			3:
				IF	(* Zylinder ist ausgefahren *)
					(e_sensor1_ausgefahren AND NOT e_sensor1_eingefahren AND NOT e_sensor_mittegefahren) OR
					(* Zylinder steht in Mittelstellung *)
					(e_sensor_mittegefahren AND NOT e_sensor1_eingefahren AND NOT e_sensor1_ausgefahren)
					THEN
						fb_state_entry.i16_next_step := AUSGEFAHREN;
				ELSE
					IF i16_betriebsart <> HAND AND st_config.b_aktiv THEN
						(* Zeitüberwachung *)
						IF fb_ton_uz_fahren.Q AND (NOT b_nockengesteuert OR b_no_gesteuert_im_norm_betrieb) THEN
							st_sm.b_zeit_ausfahren1 := TRUE;
							fb_state_entry.i16_next_step := ZYL_FEHLER;
						(* Winkelüberwachung *)
						ELSIF uw_nocken_zylinder_ausfahren AND b_nockengesteuert AND NOT b_no_gesteuert_im_norm_betrieb AND NOT b_zustand_uw_nocken_ausfahren THEN
							st_sm.b_winkel_ausfahren1 := TRUE;
							fb_state_entry.i16_next_step := ZYL_FEHLER;
						END_IF
					END_IF
				END_IF
				IF i16_betriebsart <> HAND AND st_config.b_aktiv THEN
					(* Überwachung auf Sensorfehler *)
					IF e_sensor1_ausgefahren  AND e_sensor1_eingefahren  AND st_config.b_sensor1_aktiv THEN
						fb_ton_uz_sensor1.IN := TRUE;
						IF fb_ton_uz_sensor1.Q THEN
							st_sm.b_sensor1 := TRUE;
							fb_state_entry.i16_next_step := ZYL_FEHLER;
						END_IF
					ELSE
						fb_ton_uz_sensor1.IN := FALSE;
					END_IF
				END_IF

			4:
				IF e_sensor1_ausgefahren AND e_sensor2_ausgefahren AND NOT e_sensor1_eingefahren AND NOT e_sensor2_eingefahren	THEN
					fb_state_entry.i16_next_step := AUSGEFAHREN;
				ELSE
					IF i16_betriebsart <> HAND AND st_config.b_aktiv THEN
						IF NOT e_sensor1_ausgefahren OR NOT e_sensor2_ausgefahren THEN
							(* Zeitüberwachung *)
							IF fb_ton_uz_fahren.Q AND (NOT b_nockengesteuert OR b_no_gesteuert_im_norm_betrieb) THEN
								IF NOT e_sensor1_ausgefahren THEN
									st_sm.b_zeit_ausfahren1 := TRUE;
								END_IF
								IF NOT e_sensor2_ausgefahren THEN
									st_sm.b_zeit_ausfahren2 := TRUE;
								END_IF
								fb_state_entry.i16_next_step := ZYL_FEHLER;
							(* Winkelüberwachung *)
							ELSIF uw_nocken_zylinder_ausfahren AND b_nockengesteuert AND NOT b_no_gesteuert_im_norm_betrieb AND NOT b_zustand_uw_nocken_ausfahren THEN
								IF NOT e_sensor1_ausgefahren THEN
									st_sm.b_winkel_ausfahren1 := TRUE;
								END_IF
								IF NOT e_sensor2_ausgefahren THEN
									st_sm.b_winkel_ausfahren2 := TRUE;
								END_IF
								fb_state_entry.i16_next_step := ZYL_FEHLER;
							END_IF
						END_IF
					END_IF
				END_IF

				IF i16_betriebsart <> HAND AND st_config.b_aktiv THEN
					(* Überwachung auf Sensorfehler *)
					IF e_sensor1_ausgefahren  AND e_sensor1_eingefahren  AND st_config.b_sensor1_aktiv THEN
						fb_ton_uz_sensor1.IN := TRUE;
						IF fb_ton_uz_sensor1.Q THEN
							st_sm.b_sensor1 := TRUE;
							fb_state_entry.i16_next_step := ZYL_FEHLER;
						END_IF
					ELSE
						fb_ton_uz_sensor1.IN := FALSE;
					END_IF
					IF e_sensor2_ausgefahren  AND e_sensor2_eingefahren  AND st_config.b_sensor2_aktiv THEN
						fb_ton_uz_sensor2.IN := TRUE;
						IF fb_ton_uz_sensor2.Q THEN
							st_sm.b_sensor2 := TRUE;
							fb_state_entry.i16_next_step := ZYL_FEHLER;
						END_IF
					ELSE
						fb_ton_uz_sensor2.IN := FALSE;
					END_IF
				END_IF

			6:
				IF 	e_sensor1_ausgefahren AND
					e_sensor2_ausgefahren AND
					e_sensor3_ausgefahren AND
					NOT e_sensor1_eingefahren AND
					NOT e_sensor2_eingefahren AND
					NOT e_sensor3_eingefahren
					THEN
						fb_state_entry.i16_next_step := AUSGEFAHREN;
				ELSE
					IF i16_betriebsart <> HAND AND st_config.b_aktiv THEN
						IF NOT e_sensor1_ausgefahren OR NOT e_sensor2_ausgefahren OR NOT e_sensor3_ausgefahren THEN
							(* Zeitüberwachung *)
							IF fb_ton_uz_fahren.Q AND (NOT b_nockengesteuert OR b_no_gesteuert_im_norm_betrieb) THEN
								IF NOT e_sensor1_ausgefahren THEN
									st_sm.b_zeit_ausfahren1 := TRUE;
								END_IF
								IF NOT e_sensor2_ausgefahren THEN
									st_sm.b_zeit_ausfahren2 := TRUE;
								END_IF
								IF NOT e_sensor3_ausgefahren THEN
									st_sm.b_zeit_ausfahren3 := TRUE;
								END_IF
								fb_state_entry.i16_next_step := ZYL_FEHLER;
							(* Winkelüberwachung *)
							ELSIF uw_nocken_zylinder_ausfahren AND b_nockengesteuert AND NOT b_no_gesteuert_im_norm_betrieb AND NOT b_zustand_uw_nocken_ausfahren THEN
								IF NOT e_sensor1_ausgefahren THEN
									st_sm.b_winkel_ausfahren1 := TRUE;
								END_IF
								IF NOT e_sensor2_ausgefahren THEN
									st_sm.b_winkel_ausfahren2 := TRUE;
								END_IF
								IF NOT e_sensor3_ausgefahren THEN
									st_sm.b_winkel_ausfahren3 := TRUE;
								END_IF
								fb_state_entry.i16_next_step := ZYL_FEHLER;
							END_IF
						END_IF
					END_IF
				END_IF

				IF i16_betriebsart <> HAND AND st_config.b_aktiv THEN
					(* Überwachung auf Sensorfehler *)
					IF e_sensor1_ausgefahren  AND e_sensor1_eingefahren  AND st_config.b_sensor1_aktiv THEN
						fb_ton_uz_sensor1.IN := TRUE;
						IF fb_ton_uz_sensor1.Q THEN
							st_sm.b_sensor1 := TRUE;
							fb_state_entry.i16_next_step := ZYL_FEHLER;
						END_IF
					ELSE
						fb_ton_uz_sensor1.IN := FALSE;
					END_IF
					IF e_sensor2_ausgefahren  AND e_sensor2_eingefahren  AND st_config.b_sensor2_aktiv THEN
						fb_ton_uz_sensor2.IN := TRUE;
						IF fb_ton_uz_sensor2.Q THEN
							st_sm.b_sensor2 := TRUE;
							fb_state_entry.i16_next_step := ZYL_FEHLER;
						END_IF
					ELSE
						fb_ton_uz_sensor2.IN := FALSE;
					END_IF
					IF e_sensor3_ausgefahren  AND e_sensor3_eingefahren  AND st_config.b_sensor3_aktiv THEN
						fb_ton_uz_sensor3.IN := TRUE;
						IF fb_ton_uz_sensor3.Q THEN
							st_sm.b_sensor3 := TRUE;
							fb_state_entry.i16_next_step := ZYL_FEHLER;
						END_IF
					ELSE
						fb_ton_uz_sensor3.IN := FALSE;
					END_IF
				END_IF
		END_CASE

(*=======================================================*)
	AUSGEFAHREN:
		IF fb_state_entry.E THEN
			st_ctrl_out.b_gestoppt := FALSE;
			st_ctrl_out.b_eingefahren := FALSE;
			st_ctrl_out.b_ohne_luft := FALSE;
			fb_ton_einausfahren.IN := FALSE;
			fb_ton_uz_fahren.IN := FALSE;
			fb_ton_uz_sensor1.IN := FALSE;
			fb_ton_uz_sensor2.IN := FALSE;
			fb_ton_uz_sensor3.IN := FALSE;
			st_tzk.fb_ton_tzk.IN := FALSE;
			a_ventil_ausfahren := TRUE;
			b_zustand_uw_nocken_ausfahren := FALSE;
			IF NOT b_mit_tzk THEN
				st_ctrl_out.b_ausgefahren := TRUE;
			END_IF
		END_IF

		IF st_ctrl_in.b_ausfahren THEN	(* Messagewiederholung wenn der Zylinder sich schon im gewünschten Zustand befindet*)
			st_ctrl_out.b_ausgefahren := TRUE;
		END_IF

		(*-----------------------Weiterschaltbedingungen----------------------------*)
		CASE i16_betriebsart OF
		KEINE:
			;
		AUTO, TIPPEN, DUMMY, PSEUDO:
			IF	(st_ctrl_in.b_einfahren AND
				NOT bw_nocken_zylinder_einfahren AND
				NOT b_ibn_zylinder_einfahren AND
				NOT b_direkttaste_einfahren AND
				NOT e_taste_einfahren) OR
				(NOT st_ctrl_in.b_einfahren AND
				bw_nocken_zylinder_einfahren AND
				NOT b_ibn_zylinder_einfahren AND
				NOT b_direkttaste_einfahren AND
				NOT e_taste_einfahren) OR
				(NOT st_ctrl_in.b_einfahren AND
				NOT bw_nocken_zylinder_einfahren AND
				b_ibn_zylinder_einfahren AND
				NOT b_direkttaste_einfahren AND
				NOT e_taste_einfahren)
				THEN
					IF i16_anzahl_sensoren >= 1AND b_sensor_eingefahren_vorhanden AND b_mit_tzk THEN
						st_tzk.t_einfahrzeit_kompensiert := (st_tzk.t_einfahrzeit * st_config.i16_tzk_faktor_einfahren) / 100;
					END_IF
					fb_state_entry.i16_next_step := BEWEGUNG_EINFAHREN;

			ELSIF	st_ctrl_in.b_luftlos AND
					NOT bw_nocken_zylinder_einfahren AND
					NOT b_ibn_zylinder_einfahren AND
					NOT b_direkttaste_einfahren AND
					NOT e_taste_einfahren AND
					NOT bw_nocken_zylinder_ausfahren AND
					NOT b_ibn_zylinder_ausfahren AND
					NOT b_direkttaste_ausfahren AND
					NOT e_taste_ausfahren
					THEN
						fb_state_entry.i16_next_step := LUFTLOS;
			END_IF
		HAND:
			IF	(st_visu.i16_nr_zyl_im_handbetrieb = st_config.i16_identnummer AND (st_visu.b_taste_einfahren OR e_taste_einfahren)) OR
				(bw_nocken_zylinder_einfahren AND b_nockengesteuert AND b_masterachse_hand_dialog_aktiv)
				THEN
					IF i16_anzahl_sensoren >= 1AND b_sensor_eingefahren_vorhanden AND b_mit_tzk THEN
						st_tzk.t_einfahrzeit_kompensiert := (st_tzk.t_einfahrzeit * st_config.i16_tzk_faktor_einfahren) / 100;
					END_IF
					fb_state_entry.i16_next_step := BEWEGUNG_EINFAHREN;
			END_IF
		END_CASE

		(* Überwachung auf Endlagenfehler *)
		IF i16_betriebsart <> HAND AND st_config.b_aktiv THEN
			CASE i16_anzahl_sensoren OF
				1,2,3:	(* Alle Zylinder mit mindestens einem Sensor für EINGEFAHREN *)
					IF b_sensor_ausgefahren_vorhanden AND st_config.b_endlage1_aktiv AND NOT e_sensor1_ausgefahren THEN
						fb_ton_uz_endlage1.IN := TRUE;
						IF fb_ton_uz_endlage1.Q THEN
							st_sm.b_endlage1 := TRUE;
							fb_state_entry.i16_next_step := ZYL_FEHLER;
						END_IF
					ELSE
						fb_ton_uz_endlage1.IN := FALSE;
					END_IF

				4:	(* Alle Zylinder mit 2 Sensoren für EINGEFAHREN *)
					IF b_sensor_ausgefahren_vorhanden AND st_config.b_endlage1_aktiv AND NOT e_sensor1_ausgefahren THEN
						fb_ton_uz_endlage1.IN := TRUE;
						IF fb_ton_uz_endlage1.Q THEN
							st_sm.b_endlage1 := TRUE;
							fb_state_entry.i16_next_step := ZYL_FEHLER;
						END_IF
					ELSE
						fb_ton_uz_endlage1.IN := FALSE;
					END_IF
					IF b_sensor_ausgefahren_vorhanden AND st_config.b_endlage2_aktiv AND NOT e_sensor2_ausgefahren THEN
						fb_ton_uz_endlage2.IN := TRUE;
						IF fb_ton_uz_endlage2.Q THEN
							st_sm.b_endlage2 := TRUE;
							fb_state_entry.i16_next_step := ZYL_FEHLER;
						END_IF
					ELSE
						fb_ton_uz_endlage2.IN := FALSE;
					END_IF

				6:	(* Alle Zylinder mit 3 Sensoren für EINGEFAHREN *)
					IF b_sensor_ausgefahren_vorhanden AND st_config.b_endlage1_aktiv AND NOT e_sensor1_ausgefahren THEN
						fb_ton_uz_endlage1.IN := TRUE;
						IF fb_ton_uz_endlage1.Q THEN
							st_sm.b_endlage1 := TRUE;
							fb_state_entry.i16_next_step := ZYL_FEHLER;
						END_IF
					ELSE
						fb_ton_uz_endlage1.IN := FALSE;
					END_IF
					IF b_sensor_ausgefahren_vorhanden AND st_config.b_endlage2_aktiv AND NOT e_sensor2_ausgefahren THEN
						fb_ton_uz_endlage2.IN := TRUE;
						IF fb_ton_uz_endlage2.Q THEN
							st_sm.b_endlage2 := TRUE;
							fb_state_entry.i16_next_step := ZYL_FEHLER;
						END_IF
					ELSE
						fb_ton_uz_endlage2.IN := FALSE;
					END_IF
					IF b_sensor_ausgefahren_vorhanden AND st_config.b_endlage3_aktiv AND NOT e_sensor3_ausgefahren THEN
						fb_ton_uz_endlage3.IN := TRUE;
						IF fb_ton_uz_endlage3.Q THEN
							st_sm.b_endlage3 := TRUE;
							fb_state_entry.i16_next_step := ZYL_FEHLER;
						END_IF
					ELSE
						fb_ton_uz_endlage3.IN := FALSE;
					END_IF
			END_CASE
		END_IF

(*=======================================================*)
	BEWEGUNG_EINFAHREN:
		IF fb_state_entry.E THEN
			st_ctrl_out.b_gestoppt := FALSE;
			st_ctrl_out.b_eingefahren := FALSE;
			st_ctrl_out.b_ausgefahren := FALSE;
			st_ctrl_out.b_ohne_luft := FALSE;
			st_ctrl_out.b_fehler := FALSE;
			a_ventil_ausfahren := FALSE;
			a_ventil_einfahren := TRUE;
			fb_ton_uz_fahren.IN := TRUE;
			fb_ton_einausfahren.IN := TRUE;
			fb_ton_uz_endlage1.IN := FALSE;
			fb_ton_uz_endlage2.IN := FALSE;
			fb_ton_uz_endlage3.IN := FALSE;
			st_sm.b_zeit_ausfahren1:= FALSE;
			st_sm.b_zeit_einfahren1:= FALSE;
			st_sm.b_endlage1	:= FALSE;
			st_sm.b_sensor1:= FALSE;
			st_sm.b_zeit_ausfahren2 := FALSE;
			st_sm.b_zeit_einfahren2 := FALSE;
			st_sm.b_endlage2	:= FALSE;
			st_sm.b_sensor2 := FALSE;
			st_sm.b_zeit_ausfahren3 := FALSE;
			st_sm.b_zeit_einfahren3 := FALSE;
			st_sm.b_endlage3	:= FALSE;
			st_sm.b_sensor3 := FALSE;
			st_sm.b_winkel_ausfahren1:= FALSE;
			st_sm.b_winkel_einfahren1:= FALSE;
			st_sm.b_winkel_ausfahren2 := FALSE;
			st_sm.b_winkel_einfahren2 := FALSE;
			st_sm.b_winkel_ausfahren3 := FALSE;
			st_sm.b_winkel_einfahren3 := FALSE;
			st_sm.b_zyltyp_nicht_definiert := FALSE;
			st_sm.b_reserve1:= FALSE;
			(* Verhindere die sofortige Fehlerauslösung, wenn Überwachungsnocken bei Stateentry schon vorhanden ist *)
			IF uw_nocken_zylinder_einfahren THEN
				b_zustand_uw_nocken_einfahren := TRUE;
			END_IF
		END_IF

		(* Fehlermeldung für nockengesteuerte Zylinder wieder freischalten *)
		IF fb_ton_uz_fahren.Q THEN
			b_zustand_uw_nocken_einfahren := FALSE;
		END_IF

		CASE i16_betriebsart OF
		KEINE:
			;
		AUTO, TIPPEN, DUMMY, PSEUDO:
			IF 	(st_ctrl_in.b_ausfahren AND
				NOT bw_nocken_zylinder_ausfahren AND
				NOT b_ibn_zylinder_ausfahren AND
				NOT b_direkttaste_ausfahren AND
				NOT e_taste_ausfahren) OR
				(NOT st_ctrl_in.b_ausfahren AND
				bw_nocken_zylinder_ausfahren AND
				NOT b_ibn_zylinder_ausfahren AND
				NOT b_direkttaste_ausfahren AND
				NOT e_taste_ausfahren) OR
				(NOT st_ctrl_in.b_ausfahren AND
				NOT bw_nocken_zylinder_ausfahren AND
				b_ibn_zylinder_ausfahren AND
				NOT b_direkttaste_ausfahren AND
				NOT e_taste_ausfahren)
				THEN
					IF i16_anzahl_sensoren >= 1AND b_sensor_ausgefahren_vorhanden AND b_mit_tzk THEN
						st_tzk.t_ausfahrzeit_kompensiert := (st_tzk.t_ausfahrzeit * st_config.i16_tzk_faktor_ausfahren) / 100;
					END_IF
					fb_state_entry.i16_next_step := BEWEGUNG_AUSFAHREN;
			END_IF
		HAND:
			IF	(st_visu.i16_nr_zyl_im_handbetrieb = st_config.i16_identnummer AND (st_visu.b_taste_ausfahren OR e_taste_ausfahren)) OR
				(bw_nocken_zylinder_ausfahren AND b_nockengesteuert AND b_masterachse_hand_dialog_aktiv)
				THEN
					IF i16_anzahl_sensoren >= 1AND b_sensor_ausgefahren_vorhanden AND b_mit_tzk THEN
						st_tzk.t_ausfahrzeit_kompensiert := (st_tzk.t_ausfahrzeit * st_config.i16_tzk_faktor_ausfahren) / 100;
					END_IF
					fb_state_entry.i16_next_step := BEWEGUNG_AUSFAHREN;
			END_IF
		END_CASE

		(* Totzeitkompensation mit Plausibilitätscheck der ermittelten Kompensationszeit *)
		IF 	i16_anzahl_sensoren >= 1AND
			b_sensor_eingefahren_vorhanden AND
			b_mit_tzk AND
			st_tzk.t_einfahrzeit_kompensiert < st_tzk.t_einfahrzeit
			THEN
				st_tzk.fb_ton_tzk.PT := st_tzk.t_einfahrzeit_kompensiert ;
				st_tzk.fb_ton_tzk.IN := TRUE;
				(* Totzeit ist abgelaufen -> vorzeitig "eingefahren" melden*)
				IF st_tzk.fb_ton_tzk.Q THEN
					st_tzk.fb_ton_tzk.IN := FALSE;
					st_ctrl_out.b_eingefahren := TRUE;
				END_IF
		END_IF

		(*-----------------------Weiterschaltbedingungen----------------------------*)
		(* Bedingungen für Zylinder ist eingefahren und Fehlervorkommen*)
		(* Die Sensorkonfiguration "vorhanden" ist nur für die Fälle 1, 2 von Bedeutung wegen Sonderzylinder *)
		CASE i16_anzahl_sensoren OF
			0:
				IF fb_ton_einausfahren.Q THEN
					fb_state_entry.i16_next_step := EINGEFAHREN;
				END_IF

			1:
				IF b_sensor_eingefahren_vorhanden THEN
					IF e_sensor1_eingefahren THEN
						fb_state_entry.i16_next_step := EINGEFAHREN;
					ELSE
						IF i16_betriebsart <> HAND AND st_config.b_aktiv THEN
							(* Zeitüberwachung *)
							IF fb_ton_uz_fahren.Q AND (NOT b_nockengesteuert OR b_no_gesteuert_im_norm_betrieb)THEN
								st_sm.b_zeit_einfahren1 := TRUE;
								fb_state_entry.i16_next_step := ZYL_FEHLER;
							(* Winkelüberwachung *)
							ELSIF uw_nocken_zylinder_einfahren AND b_nockengesteuert AND NOT b_no_gesteuert_im_norm_betrieb AND NOT b_zustand_uw_nocken_einfahren THEN
								st_sm.b_winkel_einfahren1 := TRUE;
								fb_state_entry.i16_next_step := ZYL_FEHLER;
							END_IF
						END_IF
					END_IF
				ELSIF b_sensor_ausgefahren_vorhanden THEN
					IF  NOT e_sensor1_ausgefahren THEN
						fb_state_entry.i16_next_step := EINGEFAHREN;
					ELSE
						IF i16_betriebsart <> HAND AND st_config.b_aktiv THEN
							(* Zeitüberwachung *)
							IF fb_ton_uz_fahren.Q AND (NOT b_nockengesteuert OR b_no_gesteuert_im_norm_betrieb)THEN
								st_sm.b_zeit_einfahren1 := TRUE;
								fb_state_entry.i16_next_step := ZYL_FEHLER;
							(* Winkelüberwachung *)
							ELSIF uw_nocken_zylinder_einfahren AND b_nockengesteuert AND NOT b_no_gesteuert_im_norm_betrieb AND NOT b_zustand_uw_nocken_einfahren THEN
								st_sm.b_winkel_einfahren1 := TRUE;
								fb_state_entry.i16_next_step := ZYL_FEHLER;
							END_IF
						END_IF
					END_IF
				END_IF

			2:
				IF b_sensor_eingefahren_vorhanden AND b_sensor_ausgefahren_vorhanden THEN
					IF e_sensor1_eingefahren AND NOT e_sensor1_ausgefahren THEN
						fb_state_entry.i16_next_step := EINGEFAHREN;
					ELSE
						IF i16_betriebsart <> HAND AND st_config.b_aktiv THEN
							(* Zeitüberwachung *)
							IF fb_ton_uz_fahren.Q AND (NOT b_nockengesteuert OR b_no_gesteuert_im_norm_betrieb)THEN
								st_sm.b_zeit_einfahren1 := TRUE;
								fb_state_entry.i16_next_step := ZYL_FEHLER;
							(* Winkelüberwachung *)
							ELSIF uw_nocken_zylinder_einfahren AND b_nockengesteuert AND NOT b_no_gesteuert_im_norm_betrieb AND NOT b_zustand_uw_nocken_einfahren THEN
								st_sm.b_winkel_einfahren1 := TRUE;
								fb_state_entry.i16_next_step := ZYL_FEHLER;
							END_IF
						END_IF
					END_IF
				ELSIF b_sensor_ausgefahren_vorhanden THEN
					IF NOT e_sensor1_ausgefahren AND NOT e_sensor2_ausgefahren THEN
						fb_state_entry.i16_next_step := EINGEFAHREN;
					ELSE
						IF i16_betriebsart <> HAND AND st_config.b_aktiv THEN
							(* Zeitüberwachung *)
							IF fb_ton_uz_fahren.Q AND (NOT b_nockengesteuert OR b_no_gesteuert_im_norm_betrieb)THEN
								IF e_sensor1_ausgefahren THEN
									st_sm.b_zeit_einfahren1 := TRUE;
								END_IF
								IF e_sensor2_ausgefahren THEN
									st_sm.b_zeit_einfahren2 := TRUE;
								END_IF
								fb_state_entry.i16_next_step := ZYL_FEHLER;
							(* Winkelüberwachung *)
							ELSIF uw_nocken_zylinder_einfahren AND b_nockengesteuert AND NOT b_no_gesteuert_im_norm_betrieb AND NOT b_zustand_uw_nocken_einfahren THEN
								IF e_sensor1_ausgefahren THEN
								st_sm.b_winkel_einfahren1 := TRUE;
								END_IF
								IF e_sensor2_ausgefahren THEN
								st_sm.b_winkel_einfahren2 := TRUE;
								END_IF
								fb_state_entry.i16_next_step := ZYL_FEHLER;
							END_IF
						END_IF
					END_IF
				ELSIF  b_sensor_eingefahren_vorhanden THEN
					IF e_sensor1_eingefahren AND e_sensor2_eingefahren THEN
						fb_state_entry.i16_next_step := EINGEFAHREN;
					ELSE
						IF i16_betriebsart <> HAND AND st_config.b_aktiv THEN
							(* Zeitüberwachung *)
							IF fb_ton_uz_fahren.Q AND (NOT b_nockengesteuert OR b_no_gesteuert_im_norm_betrieb)THEN
								IF NOT e_sensor1_eingefahren THEN
									st_sm.b_zeit_einfahren1 := TRUE;
								END_IF
								IF NOT e_sensor2_eingefahren THEN
									st_sm.b_zeit_einfahren2 := TRUE;
								END_IF
								fb_state_entry.i16_next_step := ZYL_FEHLER;
							(* Winkelüberwachung *)
							ELSIF uw_nocken_zylinder_einfahren AND b_nockengesteuert AND NOT b_no_gesteuert_im_norm_betrieb AND NOT b_zustand_uw_nocken_einfahren THEN
								IF NOT e_sensor1_eingefahren THEN
									st_sm.b_winkel_einfahren1 := TRUE;
								END_IF
								IF NOT e_sensor2_eingefahren THEN
									st_sm.b_winkel_einfahren2 := TRUE;
								END_IF
								fb_state_entry.i16_next_step := ZYL_FEHLER;
							END_IF
						END_IF
					END_IF
				END_IF
				IF i16_betriebsart <> HAND AND st_config.b_aktiv THEN
					(* Überwachung auf Sensorfehler *)
					IF e_sensor1_ausgefahren  AND e_sensor1_eingefahren  AND st_config.b_sensor1_aktiv THEN
						fb_ton_uz_sensor1.IN := TRUE;
						IF fb_ton_uz_sensor1.Q THEN
							st_sm.b_sensor1 := TRUE;
							fb_state_entry.i16_next_step := ZYL_FEHLER;
						END_IF
					ELSE
						fb_ton_uz_sensor1.IN := FALSE;
					END_IF
				END_IF

			3:
				IF	(* Zylinder ist ausgefahren *)
					(e_sensor1_eingefahren AND NOT e_sensor1_ausgefahren AND NOT e_sensor_mittegefahren) OR
					(* Zylinder steht in Mittelstellung *)
					(e_sensor_mittegefahren AND NOT e_sensor1_eingefahren AND NOT e_sensor1_ausgefahren)
					THEN
						fb_state_entry.i16_next_step := EINGEFAHREN;
				ELSE
					IF i16_betriebsart <> HAND AND st_config.b_aktiv THEN
						(* Zeitüberwachung *)
						IF fb_ton_uz_fahren.Q AND (NOT b_nockengesteuert OR b_no_gesteuert_im_norm_betrieb)THEN
							st_sm.b_zeit_einfahren1 := TRUE;
							fb_state_entry.i16_next_step := ZYL_FEHLER;
						(* Winkelüberwachung *)
						ELSIF uw_nocken_zylinder_einfahren AND b_nockengesteuert AND NOT b_no_gesteuert_im_norm_betrieb AND NOT b_zustand_uw_nocken_einfahren THEN
							st_sm.b_winkel_einfahren1 := TRUE;
							fb_state_entry.i16_next_step := ZYL_FEHLER;
						END_IF
					END_IF
				END_IF
				IF i16_betriebsart <> HAND AND st_config.b_aktiv THEN
					(* Überwachung auf Sensorfehler *)
					IF e_sensor1_ausgefahren  AND e_sensor1_eingefahren  AND st_config.b_sensor1_aktiv THEN
						fb_ton_uz_sensor1.IN := TRUE;
						IF fb_ton_uz_sensor1.Q THEN
							st_sm.b_sensor1 := TRUE;
							fb_state_entry.i16_next_step := ZYL_FEHLER;
						END_IF
					ELSE
						fb_ton_uz_sensor1.IN := FALSE;
					END_IF
				END_IF

			4:
				IF e_sensor1_eingefahren AND e_sensor2_eingefahren AND NOT e_sensor1_ausgefahren AND NOT e_sensor2_ausgefahren	THEN
					fb_state_entry.i16_next_step := EINGEFAHREN;
				ELSE
					IF i16_betriebsart <> HAND AND st_config.b_aktiv THEN
						IF NOT e_sensor1_eingefahren OR NOT e_sensor2_eingefahren THEN
							(* Zeitüberwachung *)
							IF fb_ton_uz_fahren.Q AND (NOT b_nockengesteuert OR b_no_gesteuert_im_norm_betrieb)THEN
								IF NOT e_sensor1_eingefahren THEN
									st_sm.b_zeit_einfahren1 := TRUE;
								END_IF
								IF NOT e_sensor2_eingefahren THEN
									st_sm.b_zeit_einfahren2 := TRUE;
								END_IF
								fb_state_entry.i16_next_step := ZYL_FEHLER;
							(* Winkelüberwachung *)
							ELSIF uw_nocken_zylinder_einfahren AND b_nockengesteuert AND NOT b_no_gesteuert_im_norm_betrieb AND NOT b_zustand_uw_nocken_einfahren THEN
								IF NOT e_sensor1_eingefahren THEN
									st_sm.b_winkel_einfahren1 := TRUE;
								END_IF
								IF NOT e_sensor2_eingefahren THEN
									st_sm.b_winkel_einfahren2 := TRUE;
								END_IF
								fb_state_entry.i16_next_step := ZYL_FEHLER;
							END_IF
						END_IF
					END_IF
				END_IF

				IF i16_betriebsart <> HAND AND st_config.b_aktiv THEN
					(* Überwachung auf Sensorfehler *)
					IF e_sensor1_ausgefahren  AND e_sensor1_eingefahren  AND st_config.b_sensor1_aktiv THEN
						fb_ton_uz_sensor1.IN := TRUE;
						IF fb_ton_uz_sensor1.Q THEN
							st_sm.b_sensor1 := TRUE;
							fb_state_entry.i16_next_step := ZYL_FEHLER;
						END_IF
					ELSE
						fb_ton_uz_sensor1.IN := FALSE;
					END_IF
					IF e_sensor2_ausgefahren  AND e_sensor2_eingefahren  AND st_config.b_sensor2_aktiv THEN
						fb_ton_uz_sensor2.IN := TRUE;
						IF fb_ton_uz_sensor2.Q THEN
							st_sm.b_sensor2 := TRUE;
							fb_state_entry.i16_next_step := ZYL_FEHLER;
						END_IF
					ELSE
						fb_ton_uz_sensor2.IN := FALSE;
					END_IF
				END_IF

			6:
				IF 	e_sensor1_eingefahren AND
					e_sensor2_eingefahren AND
					e_sensor3_eingefahren AND
					NOT e_sensor1_ausgefahren AND
					NOT e_sensor2_ausgefahren AND
					NOT e_sensor3_ausgefahren
					THEN
						fb_state_entry.i16_next_step := EINGEFAHREN;
				ELSE
					IF i16_betriebsart <> HAND AND st_config.b_aktiv THEN
						IF NOT e_sensor1_eingefahren OR NOT e_sensor2_eingefahren OR NOT e_sensor3_eingefahren THEN
							(* Zeitüberwachung *)
							IF fb_ton_uz_fahren.Q AND (NOT b_nockengesteuert OR b_no_gesteuert_im_norm_betrieb)THEN
								IF NOT e_sensor1_eingefahren THEN
									st_sm.b_zeit_einfahren1 := TRUE;
								END_IF
								IF NOT e_sensor2_eingefahren THEN
									st_sm.b_zeit_einfahren2 := TRUE;
								END_IF
								IF NOT e_sensor3_eingefahren THEN
									st_sm.b_zeit_einfahren3 := TRUE;
								END_IF
								fb_state_entry.i16_next_step := ZYL_FEHLER;
							(* Winkelüberwachung *)
							ELSIF uw_nocken_zylinder_einfahren AND b_nockengesteuert AND NOT b_no_gesteuert_im_norm_betrieb AND NOT b_zustand_uw_nocken_einfahren THEN
								IF NOT e_sensor1_eingefahren THEN
									st_sm.b_winkel_einfahren1 := TRUE;
								END_IF
								IF NOT e_sensor2_eingefahren THEN
									st_sm.b_winkel_einfahren2 := TRUE;
								END_IF
								IF NOT e_sensor3_eingefahren THEN
									st_sm.b_winkel_einfahren3 := TRUE;
								END_IF
								fb_state_entry.i16_next_step := ZYL_FEHLER;
							END_IF
						END_IF
					END_IF
				END_IF

				IF i16_betriebsart <> HAND AND st_config.b_aktiv THEN
					(* Überwachung auf Sensorfehler *)
					IF e_sensor1_ausgefahren  AND e_sensor1_eingefahren  AND st_config.b_sensor1_aktiv THEN
						fb_ton_uz_sensor1.IN := TRUE;
						IF fb_ton_uz_sensor1.Q THEN
							st_sm.b_sensor1 := TRUE;
							fb_state_entry.i16_next_step := ZYL_FEHLER;
						END_IF
					ELSE
						fb_ton_uz_sensor1.IN := FALSE;
					END_IF
					IF e_sensor2_ausgefahren  AND e_sensor2_eingefahren  AND st_config.b_sensor2_aktiv THEN
						fb_ton_uz_sensor2.IN := TRUE;
						IF fb_ton_uz_sensor2.Q THEN
							st_sm.b_sensor2 := TRUE;
							fb_state_entry.i16_next_step := ZYL_FEHLER;
						END_IF
					ELSE
						fb_ton_uz_sensor2.IN := FALSE;
					END_IF
					IF e_sensor3_ausgefahren  AND e_sensor3_eingefahren  AND st_config.b_sensor3_aktiv THEN
						fb_ton_uz_sensor3.IN := TRUE;
						IF fb_ton_uz_sensor3.Q THEN
							st_sm.b_sensor3 := TRUE;
							fb_state_entry.i16_next_step := ZYL_FEHLER;
						END_IF
					ELSE
						fb_ton_uz_sensor3.IN := FALSE;
					END_IF
				END_IF
		END_CASE

(*=======================================================*)
	LUFTLOS:
		IF fb_state_entry.E THEN
			a_ventil_ausfahren := FALSE;
			a_ventil_einfahren	:= FALSE;
			st_ctrl_out.b_gestoppt := FALSE;
			st_ctrl_out.b_ohne_luft := TRUE;
			st_ctrl_out.b_fehler := FALSE;
		END_IF
(*
		(* Überwachung der Sensoren *)
		CASE i16_anzahl_sensoren OF
			0:
				;

			1:
				IF b_sensor_eingefahren_vorhanden THEN
					IF st_ctrl_out.b_eingefahren AND NOT e_sensor1_eingefahren THEN
						st_sm.b_endlage1 := TRUE;
						fb_state_entry.i16_next_step := ZYL_FEHLER;
					END_IF
				ELSIF b_sensor_ausgefahren_vorhanden THEN
					IF  st_ctrl_out.b_ausgefahren AND NOT e_sensor1_ausgefahren THEN
						st_sm.b_endlage1 := TRUE;
						fb_state_entry.i16_next_step := ZYL_FEHLER;
					END_IF
				END_IF

			2:
				IF b_sensor_eingefahren_vorhanden AND b_sensor_ausgefahren_vorhanden THEN
					IF 	(st_ctrl_out.b_eingefahren AND NOT e_sensor1_eingefahren) OR
						(st_ctrl_out.b_ausgefahren AND NOT e_sensor1_ausgefahren)
						THEN
							st_sm.b_endlage1 := TRUE;
							fb_state_entry.i16_next_step := ZYL_FEHLER;
					END_IF
				ELSIF b_sensor_ausgefahren_vorhanden THEN
					IF st_ctrl_out.b_ausgefahren AND (NOT e_sensor1_ausgefahren OR NOT e_sensor2_ausgefahren) THEN
						st_sm.b_endlage1 := NOT e_sensor1_ausgefahren;
						st_sm.b_endlage2 := NOT e_sensor2_ausgefahren;
						fb_state_entry.i16_next_step := ZYL_FEHLER;
					END_IF
				ELSIF  b_sensor_eingefahren_vorhanden THEN
					IF st_ctrl_out.b_eingefahren AND (NOT e_sensor1_eingefahren OR NOT e_sensor2_eingefahren) THEN
						st_sm.b_endlage1 := NOT e_sensor1_eingefahren;
						st_sm.b_endlage2 := NOT e_sensor2_eingefahren;
						fb_state_entry.i16_next_step := ZYL_FEHLER;
					END_IF
				END_IF

			3:
				;

			4:
				IF st_ctrl_out.b_eingefahren AND (NOT e_sensor1_eingefahren OR NOT e_sensor2_eingefahren)THEN
					st_sm.b_endlage1 := NOT e_sensor1_eingefahren;
					st_sm.b_endlage2 := NOT e_sensor2_eingefahren;
					fb_state_entry.i16_next_step := ZYL_FEHLER;
				ELSIF st_ctrl_out.b_ausgefahren AND (NOT e_sensor1_ausgefahren OR NOT e_sensor2_ausgefahren)THEN
					st_sm.b_endlage1 := NOT e_sensor1_ausgefahren;
					st_sm.b_endlage2 := NOT e_sensor2_ausgefahren;
					fb_state_entry.i16_next_step := ZYL_FEHLER;
				END_IF

			6:
				IF st_ctrl_out.b_eingefahren AND (NOT e_sensor1_eingefahren OR NOT e_sensor2_eingefahren OR NOT e_sensor3_eingefahren)THEN
					st_sm.b_endlage1 := NOT e_sensor1_eingefahren;
					st_sm.b_endlage2 := NOT e_sensor2_eingefahren;
					st_sm.b_endlage3 := NOT e_sensor3_eingefahren;
					fb_state_entry.i16_next_step := ZYL_FEHLER;
				ELSIF st_ctrl_out.b_ausgefahren AND (NOT e_sensor1_ausgefahren OR NOT e_sensor2_ausgefahren OR NOT e_sensor2_ausgefahren)THEN
					st_sm.b_endlage1 := NOT e_sensor1_ausgefahren;
					st_sm.b_endlage2 := NOT e_sensor2_ausgefahren;
					st_sm.b_endlage3 := NOT e_sensor3_ausgefahren;
					fb_state_entry.i16_next_step := ZYL_FEHLER;
				END_IF
		END_CASE
*)
		(*-----------------------Weiterschaltbedingungen----------------------------*)
		CASE i16_betriebsart OF
		KEINE:
			;
		AUTO, TIPPEN, DUMMY, PSEUDO:
			IF 	(st_ctrl_in.b_ausfahren AND
				NOT st_ctrl_in.b_luftlos AND
				NOT bw_nocken_zylinder_ausfahren AND
				NOT b_ibn_zylinder_ausfahren AND
				NOT b_direkttaste_ausfahren AND
				NOT e_taste_ausfahren) OR
				(NOT st_ctrl_in.b_ausfahren AND
				NOT st_ctrl_in.b_luftlos AND
				bw_nocken_zylinder_ausfahren AND
				NOT b_ibn_zylinder_ausfahren AND
				NOT b_direkttaste_ausfahren AND
				NOT e_taste_ausfahren) OR
				(NOT st_ctrl_in.b_ausfahren AND
				NOT st_ctrl_in.b_luftlos AND
				NOT bw_nocken_zylinder_ausfahren AND
				b_ibn_zylinder_ausfahren AND
				NOT b_direkttaste_ausfahren AND
				NOT e_taste_ausfahren)
				THEN
					fb_state_entry.i16_next_step := BEWEGUNG_AUSFAHREN;

			ELSIF	(st_ctrl_in.b_einfahren AND
					NOT st_ctrl_in.b_luftlos AND
					NOT bw_nocken_zylinder_einfahren AND
					NOT b_ibn_zylinder_einfahren AND
					NOT b_direkttaste_einfahren AND
					NOT e_taste_einfahren) OR
					(NOT st_ctrl_in.b_einfahren AND
					NOT st_ctrl_in.b_luftlos AND
					bw_nocken_zylinder_einfahren AND
					NOT b_ibn_zylinder_einfahren AND
					NOT b_direkttaste_einfahren AND
					NOT e_taste_einfahren) OR
					(NOT st_ctrl_in.b_einfahren AND
					NOT st_ctrl_in.b_luftlos AND
					NOT bw_nocken_zylinder_einfahren AND
					b_ibn_zylinder_einfahren AND
					NOT b_direkttaste_einfahren AND
					NOT e_taste_einfahren)
					THEN
						fb_state_entry.i16_next_step := BEWEGUNG_EINFAHREN;
			END_IF
		HAND:
			IF	(st_visu.i16_nr_zyl_im_handbetrieb = st_config.i16_identnummer AND (st_visu.b_taste_ausfahren OR e_taste_ausfahren)) OR
				(bw_nocken_zylinder_ausfahren AND b_nockengesteuert AND b_masterachse_hand_dialog_aktiv)
				THEN
					fb_state_entry.i16_next_step := BEWEGUNG_AUSFAHREN;

			ELSIF	(st_visu.i16_nr_zyl_im_handbetrieb = st_config.i16_identnummer AND (st_visu.b_taste_einfahren OR e_taste_einfahren)) OR
					(bw_nocken_zylinder_einfahren AND b_nockengesteuert AND b_masterachse_hand_dialog_aktiv)
					THEN
						fb_state_entry.i16_next_step := BEWEGUNG_EINFAHREN;
			END_IF
		END_CASE


(*=======================================================*)
	ZYL_FEHLER:
		IF fb_state_entry.E THEN
			st_ctrl_out.b_fehler := TRUE;
			st_ctrl_out.b_eingefahren := FALSE;
			st_ctrl_out.b_ausgefahren := FALSE;
			st_ctrl_out.b_gestoppt := FALSE;
			fb_ton_quitt.IN := FALSE;
			st_visu.i16_zyl_id := st_config.i16_identnummer;
			st_visu.i16_zyl_fehlergruppe := st_config.i16_gruppe;
		END_IF

		(* Fehler wurde quittiert *)
		IF (st_ctrl_in.b_quittieren  OR b_ibn_zylinderfehler_quit ) AND NOT fb_state_entry.E THEN
			st_ctrl_out.b_fehler := FALSE;
			fb_ton_quitt.IN := TRUE;
		END_IF

		IF fb_ton_quitt.Q THEN
			fb_ton_quitt.IN := FALSE;
			fb_state_entry.i16_next_step := ZYL_INIT;
		END_IF

		(* Weiterschaltbedingungen für das Bewegen der Zylinder im Visu-Auswahlmenü im Handbetrieb, Hardwaretaster *)
		(* Zylinder einfahren im Handbetrieb über Tasten *)
		IF	i16_betriebsart = HAND AND
			st_visu.i16_nr_zyl_im_handbetrieb = st_config.i16_identnummer AND
			st_visu.b_taste_ausfahren AND
			NOT st_visu.b_taste_einfahren
			THEN
				st_ctrl_out.b_fehler := FALSE;
				st_sm.b_zeit_ausfahren1:= FALSE;
				st_sm.b_zeit_einfahren1:= FALSE;
				st_sm.b_endlage1	:= FALSE;
				st_sm.b_sensor1:= FALSE;
				st_sm.b_zeit_ausfahren2 := FALSE;
				st_sm.b_zeit_einfahren2 := FALSE;
				st_sm.b_endlage2	:= FALSE;
				st_sm.b_sensor2 := FALSE;
				st_sm.b_zeit_ausfahren3 := FALSE;
				st_sm.b_zeit_einfahren3 := FALSE;
				st_sm.b_endlage3	:= FALSE;
				st_sm.b_sensor3 := FALSE;
				st_sm.b_winkel_ausfahren1:= FALSE;
				st_sm.b_winkel_einfahren1:= FALSE;
				st_sm.b_winkel_ausfahren2 := FALSE;
				st_sm.b_winkel_einfahren2 := FALSE;
				st_sm.b_winkel_ausfahren3 := FALSE;
				st_sm.b_winkel_einfahren3 := FALSE;
				st_sm.b_zyltyp_nicht_definiert := FALSE;
				st_sm.b_reserve1:= FALSE;
				fb_state_entry.i16_next_step := BEWEGUNG_AUSFAHREN;

		(* Zylinder einfahren im Handbetrieb über Tasten *)
		ELSIF i16_betriebsart = HAND AND
			st_visu.i16_nr_zyl_im_handbetrieb = st_config.i16_identnummer AND
			st_visu.b_taste_einfahren AND
			NOT st_visu.b_taste_ausfahren
			THEN
				st_ctrl_out.b_fehler := FALSE;
				st_sm.b_zeit_ausfahren1:= FALSE;
				st_sm.b_zeit_einfahren1:= FALSE;
				st_sm.b_endlage1	:= FALSE;
				st_sm.b_sensor1:= FALSE;
				st_sm.b_zeit_ausfahren2 := FALSE;
				st_sm.b_zeit_einfahren2 := FALSE;
				st_sm.b_endlage2	:= FALSE;
				st_sm.b_sensor2 := FALSE;
				st_sm.b_zeit_ausfahren3 := FALSE;
				st_sm.b_zeit_einfahren3 := FALSE;
				st_sm.b_endlage3	:= FALSE;
				st_sm.b_sensor3 := FALSE;
				st_sm.b_winkel_ausfahren1:= FALSE;
				st_sm.b_winkel_einfahren1:= FALSE;
				st_sm.b_winkel_ausfahren2 := FALSE;
				st_sm.b_winkel_einfahren2 := FALSE;
				st_sm.b_winkel_ausfahren3 := FALSE;
				st_sm.b_winkel_einfahren3 := FALSE;
				st_sm.b_zyltyp_nicht_definiert := FALSE;
				st_sm.b_reserve1:= FALSE;
				fb_state_entry.i16_next_step := BEWEGUNG_EINFAHREN;
		END_IF

(*=======================================================*)
	DIREKT_AUSFAHREN:
		IF fb_state_entry.E THEN
			a_ventil_ausfahren := TRUE;
			a_ventil_einfahren := FALSE;
		END_IF

		IF NOT b_direkttaste_ausfahren AND NOT e_taste_ausfahren THEN
			fb_state_entry.i16_next_step := GESTOPPT;
		END_IF

(*=======================================================*)
	DIREKT_EINFAHREN:
		IF fb_state_entry.E THEN
			a_ventil_ausfahren := FALSE;
			a_ventil_einfahren := TRUE;
		END_IF

		IF NOT b_direkttaste_einfahren AND NOT e_taste_einfahren THEN
			fb_state_entry.i16_next_step := GESTOPPT;
		END_IF
END_CASE

fb_state_entry(
	i16_next_step:= ,
	i16_pos:= 2,
	s_debugtext:= ,
	E=> , 
	X=> , 
	i16_step=> ,
	i16_last_step=> );

IF st_config.b_config_fertig THEN
	(* Fehlermeldungen und Betriebsmeldungen ab dem Startindex in die globalen Meldungsarrays schreiben *)
	garr_stoermeldungen[st_config.i16_meld_startindex + 0] := st_sm.b_zeit_ausfahren1;
	garr_stoermeldungen[st_config.i16_meld_startindex + 1] := st_sm.b_zeit_einfahren1;
	garr_stoermeldungen[st_config.i16_meld_startindex + 2] := st_sm.b_endlage1;
	garr_stoermeldungen[st_config.i16_meld_startindex + 3] := st_sm.b_sensor1;
	garr_stoermeldungen[st_config.i16_meld_startindex + 4] := st_sm.b_zeit_ausfahren2;
	garr_stoermeldungen[st_config.i16_meld_startindex + 5] := st_sm.b_zeit_einfahren2;
	garr_stoermeldungen[st_config.i16_meld_startindex + 6] := st_sm.b_endlage2;
	garr_stoermeldungen[st_config.i16_meld_startindex + 7] := st_sm.b_sensor2;
	garr_stoermeldungen[st_config.i16_meld_startindex + 8] := st_sm.b_zeit_ausfahren3;
	garr_stoermeldungen[st_config.i16_meld_startindex + 9] := st_sm.b_zeit_einfahren3;
	garr_stoermeldungen[st_config.i16_meld_startindex + 10] := st_sm.b_endlage3;
	garr_stoermeldungen[st_config.i16_meld_startindex + 11] := st_sm.b_sensor3;
	garr_stoermeldungen[st_config.i16_meld_startindex + 12] := st_sm.b_winkel_ausfahren1;
	garr_stoermeldungen[st_config.i16_meld_startindex + 13] := st_sm.b_winkel_einfahren1;
	garr_stoermeldungen[st_config.i16_meld_startindex + 14] := st_sm.b_winkel_ausfahren2;
	garr_stoermeldungen[st_config.i16_meld_startindex + 15] := st_sm.b_winkel_einfahren2;
	garr_stoermeldungen[st_config.i16_meld_startindex + 16] := st_sm.b_winkel_ausfahren3;
	garr_stoermeldungen[st_config.i16_meld_startindex + 17] := st_sm.b_winkel_einfahren3;
	garr_stoermeldungen[st_config.i16_meld_startindex + 18] := st_sm.b_zyltyp_nicht_definiert;
	garr_stoermeldungen[st_config.i16_meld_startindex + 19] := st_sm.b_reserve1;
	
	garr_betriebsmeldungen[st_config.i16_meld_startindex + 0] := FALSE;
	garr_betriebsmeldungen[st_config.i16_meld_startindex + 1] := FALSE;
	garr_betriebsmeldungen[st_config.i16_meld_startindex + 2] := FALSE;
	garr_betriebsmeldungen[st_config.i16_meld_startindex + 3] := FALSE;
	garr_betriebsmeldungen[st_config.i16_meld_startindex + 4] := FALSE;
	garr_betriebsmeldungen[st_config.i16_meld_startindex + 5] := FALSE;
	garr_betriebsmeldungen[st_config.i16_meld_startindex + 6] := FALSE;
	garr_betriebsmeldungen[st_config.i16_meld_startindex + 7] := FALSE;
	garr_betriebsmeldungen[st_config.i16_meld_startindex + 8] := FALSE;
	garr_betriebsmeldungen[st_config.i16_meld_startindex + 9] := FALSE;
	garr_betriebsmeldungen[st_config.i16_meld_startindex + 10] := FALSE;
	garr_betriebsmeldungen[st_config.i16_meld_startindex + 11] := FALSE;
	garr_betriebsmeldungen[st_config.i16_meld_startindex + 12] := FALSE;
	garr_betriebsmeldungen[st_config.i16_meld_startindex + 13] := FALSE;
	garr_betriebsmeldungen[st_config.i16_meld_startindex + 14] := FALSE;
	garr_betriebsmeldungen[st_config.i16_meld_startindex + 15] := FALSE;
	garr_betriebsmeldungen[st_config.i16_meld_startindex + 16] := FALSE;
	garr_betriebsmeldungen[st_config.i16_meld_startindex + 17] := FALSE;
	garr_betriebsmeldungen[st_config.i16_meld_startindex + 18] := FALSE;
	garr_betriebsmeldungen[st_config.i16_meld_startindex + 19] := FALSE;
END_IF
END_FUNCTION_BLOCK

(* POU Gemeinsamkeiten17xx/Allgemeines/ST_Betriebsstundenzaehler, ST *)
FUNCTION_BLOCK ST_Betriebsstundenzaehler
VAR_INPUT
	b_eingekuppelt					: BOOL;
	b_reset							: BOOL;
	i32_betriebssekundenzaehler_in		: UDINT;
END_VAR
VAR_OUTPUT
	t_betriebsstunden_neu				: TIME;
	i32_betriebssekundenzaehler 		: UDINT;
	lr_betriebsstundenzaehler 			: LREAL;
END_VAR
VAR
	b_first_cycle						: BOOL := TRUE;
	fb_ton							: TON;
	t_betriebssekunden_Merker			: TIME := t#0ms;
	a_betriebsstundenzaehler 			AT %Q* : BOOL;
END_VAR
IF b_first_cycle THEN
 	i32_betriebssekundenzaehler := i32_betriebssekundenzaehler_in;
	b_first_cycle := FALSE;
END_IF

(* Hardware-Betriebsstundenzähler *)
a_betriebsstundenzaehler := b_eingekuppelt;

IF NOT b_eingekuppelt  THEN
	t_betriebssekunden_Merker := t_betriebssekunden_Merker + fb_ton.ET;
END_IF

fb_ton(IN:=b_eingekuppelt, PT:= t#24h, Q=> , ET=> );

IF gi16_maschinenstatusinfo <> STATUS_MASCHINE_ARBEITET AND NOT b_eingekuppelt THEN
	i32_betriebssekundenzaehler:=i32_betriebssekundenzaehler + (TIME_TO_UDINT(t_betriebssekunden_Merker)/1000);
	t_betriebssekunden_Merker:=t#0ms;
END_IF

lr_betriebsstundenzaehler:=UDINT_TO_LREAL(i32_betriebssekundenzaehler) / 3600;
END_FUNCTION_BLOCK

(* POU Gemeinsamkeiten17xx/Barcode/ST_Barcode, ST *)
FUNCTION_BLOCK ST_Barcode
VAR_INPUT
	st_config					: struct_config;

	b_steuerung_ein				: BOOL;
	b_bandende_links			: BOOL;
	b_bandende_rechts			: BOOL;
	b_bandende_1720			: BOOL;
END_VAR
VAR_IN_OUT
	st_barcode_daten			: struct_barcode_daten;
END_VAR
VAR_OUTPUT
	b_band_nicht_gescannt		: BOOL;
END_VAR
VAR
	fb_state_entry				: ST_StateEntry;
	fb_ton_wz					: TON;

	fb_tof_bandende_li			: TOF;
	fb_tof_bandende_re			: TOF;
	fb_tof_bandende_1720		: TOF;

	fb_trig_LTS_aus				: R_TRIG;
	st_LTS_xml					: struct_LTS_xml;
	i_actuellVPE				: DINT;			(*Verpackungseinheit*)
	s_FileName					: STRING;

	fb_WriteXml					: FB_XmlSrvWriteByName;
	NT_StartProcess 			: NT_StartProcess;
	fb_state_entry2				: ST_StateEntry;
	i_ErrId						: UDINT;

	(* RS232-Schnittstelle *)
	(* Hinweis: Datenpuffer vom Typ ComBuffer werden vom Anwender niemals direkt beschrieben oder gelesen,
	sondern dienen nur als Zwischenspeicher für die Kommunikationsbausteine. *)
	RxBuffer						: ComBuffer;
	TxBuffer						: ComBuffer;
	COM_in_data AT %I* 			: PcComInData; (*EL6inData22B;*)
	COM_out_data AT %Q*  			: PcComOutData; (*EL6outData22B;*)
	fb_com_port_control				: SerialLineControl;
	com_port_control_error			: BOOL := FALSE;
	com_port_control_error_id		: ComError_t;

	(* ReceiveString empfängt eine Zeichenkette von der mit der Eingangsvariablen RxBuffer korrespondierenden Schnittstelle
	und speichert sie in der Ausgangsvariablen ReceivedString. *)
	fb_receive					: ReceiveString;
	fb_trig_new_string			: R_TRIG;
	s_tmp_string					: STRING := '';

	s_start_wkz					: STRING :='';
	s_start_band_links			: STRING :='';
	s_start_band_rechts			: STRING :='';
	s_start_band				: STRING :='';

	sm_fehler_seriel				: BOOL := FALSE;

	fb_tof_bm_neues_band_links		: TOF;
	fb_tof_bm_neues_band_rechts	: TOF;
	fb_tof_bm_neues_band_1720	: TOF;
	fb_tof_bm_neues_wkz			: TOF;
	fb_trig_manuell					: F_TRIG;

	bm_band_nicht_gescannt_links	: BOOL := FALSE;
	bm_band_nicht_gescannt_rechts	: BOOL := FALSE;

	s_band_anwahl_copy			: STRING;
	s_wkz_anwahl_copy				: STRING;

	i								: INT;
	m_WpcNumber_links			: BYTE;
	b_Zaehler_WPC_links			: INT;
	m_WpcNumber_rechts			: BYTE;
	b_Zaehler_WPC_rechts			: INT;
	i16_WT_auf_Band				: INT := 13;

	s_band_ID_linksHelp			: STRING(20) :='';
	s_band_ID_rechtsHelp			: STRING(20) :='';
	fb_ton_band_ID					: TON;
	b_newbatchOk					: BOOL;
END_VAR
(*
Baustein läuft fast komplett entkoppelt vom Hauptablauf. Es soll nicht der Barcodescanner zum Stop der Anlage führen.
Der restliche Ablauf greift nur über die persistenten Daten auf die "freigaben" und die angewählten Bänder zu

Funktion:
	bei Steuerung aus:
	---------------------------
		Scan Start Werkzeug, Scan Werkzeugcode ==> Anwahl des Werkzeuges
		Scan Start Band, Scan bandcode ==> Anwahl des Bandes

	bei Steuerung ein:
	---------------------------
		Scan Start Werkzeug, Scan Werkzeugcode ==> Keine Reaktion
		Scan Start Band(Links|Rechts), Scan bandcode ==> Stimmt Band mit Angewähltem Band überein, wird Band_x_ok gesetzt.

		Bandende_x = False ==> Band_x_ok wird false gesetzt
*)

fb_trig_manuell(CLK:= gst_datensatz.st_md.i16_typ_bestueckmodus = BESTUECKUNG_MANUAL, Q=> );

(* Toplevel *)
IF fb_state_entry.i16_next_step > INIT AND fb_state_entry.i16_next_step < FEHLER THEN

	IF com_port_control_error OR fb_receive.Error > 0 THEN
		sm_fehler_seriel := TRUE;
		fb_state_entry.i16_next_step := FEHLER;
	END_IF
END_IF

(* Abwahl Band ok =======================================================*)
(* Bandende entprellen *)
IF	b_steuerung_ein THEN
	fb_tof_bandende_li(IN:= b_bandende_links , PT:=t#1s , Q=>  , ET=> );
	fb_tof_bandende_re(IN:=b_bandende_rechts  , PT:=t#1s , Q=>  , ET=> );
	fb_tof_bandende_1720(IN:=b_bandende_1720 , PT:=t#1s , Q=>  , ET=> );

	IF NOT fb_tof_bandende_li.Q THEN
		st_barcode_daten.b_band_links_ok := FALSE;
		st_barcode_daten.b_band_ID_links_ok := FALSE;
		st_barcode_daten.s_band_ID_links:='';
		s_band_ID_linksHelp:='';
	END_IF
	IF NOT fb_tof_bandende_re.Q THEN
		st_barcode_daten.b_band_rechts_ok := FALSE;
		st_barcode_daten.b_band_ID_rechts_ok := FALSE;
		st_barcode_daten.s_band_ID_rechts:='';
		s_band_ID_rechtsHelp:='';
	END_IF
	IF NOT fb_tof_bandende_1720.Q AND gst_datensatz.st_md.i16_typ_zelle= BESTUECKZELLE_1720 THEN
		st_barcode_daten.b_band_ok := FALSE;
		st_barcode_daten.b_band_rechts_ok := FALSE;
		st_barcode_daten.b_band_ID_rechts_ok := FALSE;
		st_barcode_daten.s_band_ID_rechts:='';
		s_band_ID_rechtsHelp:='';
		st_barcode_daten.b_band_links_ok := FALSE;
		st_barcode_daten.b_band_ID_links_ok := FALSE;
		st_barcode_daten.s_band_ID_links:='';
		s_band_ID_linksHelp:='';
	END_IF
END_IF

(* Betriebsmeldungen wenn Band eingefädelt ist, aber nicht abgescannt *)
bm_band_nicht_gescannt_links := b_bandende_links AND (NOT st_barcode_daten.b_band_links_ok OR NOT st_barcode_daten.b_band_ID_links_ok);
bm_band_nicht_gescannt_rechts := b_bandende_rechts AND (NOT st_barcode_daten.b_band_rechts_ok OR NOT st_barcode_daten.b_band_ID_rechts_ok);
b_band_nicht_gescannt := bm_band_nicht_gescannt_links OR bm_band_nicht_gescannt_rechts; (* für Lampe Materialmangel *)

IF	gst_datensatz.st_md.b_band_ID_Puffer_aus THEN
	st_barcode_daten.b_band_ID_rechts_ok := TRUE;
	st_barcode_daten.b_band_ID_links_ok := TRUE;
ELSE
	ChargeToLTS();
END_IF

fb_trig_LTS_aus(CLK:=NOT gst_datensatz.st_md.b_band_ID_Puffer_aus);
IF	fb_trig_LTS_aus.Q THEN
	st_barcode_daten.b_band_ID_rechts_ok := FALSE;
	st_barcode_daten.b_band_ID_links_ok := FALSE;
END_IF

(*Anzeige Visu hinten für WZ und Band ================================*)
visu_hinten.in.s_aktuelles_band:=gst_datensatz.st_md.s_aktuelles_band;
visu_hinten.in.s_aktuelles_wkz:=gst_datensatz.st_md.s_aktuelles_wkz;

fb_ton_wz(IN:= , PT:=t#10s , Q=>  , ET=> );
IF	fb_trig_new_string.Q THEN
	fb_ton_wz.IN:=TRUE;
	visu_hinten.in.s_Barcode:=s_tmp_string;
END_IF
IF	fb_ton_wz.Q THEN
	fb_ton_wz.IN:=FALSE;
	visu_hinten.in.s_Barcode:='';
END_IF


(*Band scannen möglich============================================*)
IF	b_bandende_rechts  THEN
	visu_hinten.in.scannen_moeglich[0]:= TRUE;
END_IF
IF	(b_bandende_rechts AND visu_hinten.in.bandfreigabe[0] ) OR
	NOT b_bandende_rechts  OR
	NOT b_steuerung_ein THEN
	visu_hinten.in.scannen_moeglich[0]:= FALSE;
END_IF

IF	b_bandende_links  THEN
	visu_hinten.in.scannen_moeglich[1]:= TRUE;
END_IF
IF	(b_bandende_links AND visu_hinten.in.bandfreigabe[1] ) OR
	NOT b_bandende_links OR
	NOT b_steuerung_ein THEN
	visu_hinten.in.scannen_moeglich[1]:= FALSE;
END_IF

IF 	fb_trig_manuell.Q OR
	s_band_anwahl_copy<>st_barcode_daten.s_band_anwahl OR	(* Bei einer Änderung an der Visu Band OK zurücksetzen*)
	s_wkz_anwahl_copy<>st_barcode_daten.s_wkz_anwahl THEN

	s_band_anwahl_copy :=st_barcode_daten.s_band_anwahl;
	s_wkz_anwahl_copy:=st_barcode_daten.s_wkz_anwahl;
	st_barcode_daten.b_band_links_ok := FALSE;
	st_barcode_daten.b_band_rechts_ok := FALSE;
	st_barcode_daten.b_band_ok := FALSE;
	st_barcode_daten.s_band_ID_links:='';
	st_barcode_daten.b_band_ID_links_ok := FALSE;
	st_barcode_daten.s_band_ID_rechts:='';
	st_barcode_daten.b_band_ID_rechts_ok := FALSE;
	s_band_ID_linksHelp:='';
	s_band_ID_rechtsHelp:='';
END_IF

(* Meldungs TOFs *)
fb_tof_bm_neues_band_links.IN := FALSE;
fb_tof_bm_neues_band_rechts.IN := FALSE;
fb_tof_bm_neues_band_1720.IN := FALSE;
fb_tof_bm_neues_wkz.IN := FALSE;

(* ==================================Schrittkette================================ *)
fb_state_entry(i16_pos:= 1);

CASE fb_state_entry.i16_step OF
(*=======================================================*)
	INIT_OBJ:
		IF 	st_config.b_config_fertig THEN
			fb_state_entry.i16_next_step := INIT;
		END_IF

(*=======================================================*)
	INIT:
		IF 	fb_state_entry.E THEN
			sm_fehler_seriel := FALSE;

			s_start_wkz			:= 'WKZ';
			s_start_band_links	:= 'BAL';
			s_start_band_rechts	:= 'BAR';
			s_start_band		:= 'BAB';

		END_IF

		(*-----------------------Weiterschaltbedingungen----------------------------*)
			(* start verzögerung *)
		IF 	fb_state_entry.fb_ton_Step.ET > t#1s THEN
			fb_state_entry.i16_next_step := 20;
		END_IF

(*=======================================================*)
	20:  fb_state_entry.s_debugtext:='Reset Schnittstelle';

		IF 	fb_state_entry.E THEN
			fb_receive.Reset := TRUE;
		END_IF

		(*-----------------------Weiterschaltbedingungen----------------------------*)
		IF 	fb_state_entry.fb_ton_Step.ET > t#100ms THEN
			fb_receive.Reset := FALSE;
			fb_state_entry.i16_next_step := BEREIT;
		END_IF

(*=======================================================*)
	BEREIT:  fb_state_entry.s_debugtext:='Warte Ereigniss';

		IF 	st_barcode_daten.b_band_links_ok AND
			st_barcode_daten.b_band_rechts_ok THEN
			st_barcode_daten.b_band_ok := TRUE;
		ELSE
			st_barcode_daten.b_band_ok := FALSE;
		END_IF

		IF 	st_barcode_daten.s_band_anwahl <> gst_datensatz.st_md.s_aktuelles_band THEN
			(* Anwahl von Hand *)
			st_barcode_daten.s_band_anwahl := gst_datensatz.st_md.s_aktuelles_band ;
		END_IF

		IF 	st_barcode_daten.s_wkz_anwahl <> gst_datensatz.st_md.s_aktuelles_wkz THEN
			(* Anwahl von Hand *)
			 st_barcode_daten.s_wkz_anwahl := gst_datensatz.st_md.s_aktuelles_wkz;
		END_IF

		IF 	fb_trig_new_string.Q THEN
			Anwahl();
		END_IF

		HandeingabeID();

(*=======================================================*)
	200:  fb_state_entry.s_debugtext:='Werkzeug';

		IF 	fb_trig_new_string.Q THEN
			(* 23.02.22 Wunsch von D. Rustler: Barcode soll bei Steuerung aus dasselbe machen wie bei Steuerung Ein
			Also keine Werkzeuganwahl mehr *)

			(* Keine Reaktion *)
			Anwahl()
			(* Wenn nicht verzweigt wurde, wieder nach BEREIT *);
			IF fb_state_entry.i16_next_step = 200 THEN
				fb_state_entry.i16_next_step := BEREIT;
			END_IF
		END_IF

		(* Wartezeit abgelaufen => Wieder bereit *)
		IF 	fb_state_entry.fb_ton_Step.ET > t#5s THEN
 			fb_state_entry.s_debugtext:=CONCAT(fb_state_entry.s_debugtext,' => Wartezeit abgelaufen');
			fb_state_entry.i16_next_step := BEREIT;
		END_IF

(*=======================================================*)
	300:  fb_state_entry.s_debugtext:='Band Links';

		IF 	fb_trig_new_string.Q THEN
			Anwahl();
			IF 	fb_state_entry.i16_next_step = 300  AND
				s_tmp_string = st_barcode_daten.s_band_anwahl AND b_bandende_links THEN
				st_barcode_daten.b_band_links_ok := TRUE;
				fb_state_entry.i16_next_step := BEREIT;
			END_IF
		END_IF

		(* Wartezeit abgelaufen => Wieder bereit *)
		IF 	fb_state_entry.fb_ton_Step.ET > t#5s THEN
 			fb_state_entry.s_debugtext:=CONCAT(fb_state_entry.s_debugtext,' => Wartezeit abgelaufen');
			fb_state_entry.i16_next_step := BEREIT;
		END_IF

(*=======================================================*)
	350:  fb_state_entry.s_debugtext:='Band ID links';

		IF 	fb_trig_new_string.Q AND b_steuerung_ein THEN
			IF	s_tmp_string <> st_barcode_daten.s_band_anwahl AND
				s_tmp_string <> st_barcode_daten.s_band_ID_rechts AND
				b_bandende_links AND
				FIND(s_tmp_string,'-') <> 4 AND
				LEN(s_tmp_string) >8 AND
				(LEN(s_tmp_string) =10 OR gst_datensatz.st_md.i16_typ_zelle <> RASTERFOLIE) THEN
				st_barcode_daten.s_band_ID_links:=s_tmp_string;
				st_barcode_daten.b_band_ID_links_ok := TRUE;
				fb_tof_bm_neues_band_links.IN := TRUE;
				s_band_ID_linksHelp:=st_barcode_daten.s_band_ID_links;
			END_IF
			fb_state_entry.i16_next_step := BEREIT;
		END_IF

		(* Wartezeit abgelaufen => Wieder bereit *)
		IF 	fb_state_entry.fb_ton_Step.ET > t#5s THEN
 			fb_state_entry.s_debugtext:=CONCAT(fb_state_entry.s_debugtext,' => Wartezeit abgelaufen');
			fb_state_entry.i16_next_step := BEREIT;
		END_IF

(*=======================================================*)
	400:  fb_state_entry.s_debugtext:='Band Rechts';

		IF 	fb_trig_new_string.Q THEN
			Anwahl();
			IF  	fb_state_entry.i16_next_step = 400  AND s_tmp_string = st_barcode_daten.s_band_anwahl AND b_bandende_rechts THEN
				st_barcode_daten.b_band_rechts_ok := TRUE;
				fb_state_entry.i16_next_step := BEREIT;
			END_IF
		END_IF

		(* Wartezeit abgelaufen => Wieder bereit *)
		IF 	fb_state_entry.fb_ton_Step.ET > t#5s THEN
 			fb_state_entry.s_debugtext:=CONCAT(fb_state_entry.s_debugtext,' => Wartezeit abgelaufen');
			fb_state_entry.i16_next_step := BEREIT;
		END_IF

(*=======================================================*)
	450:  fb_state_entry.s_debugtext:='Band ID rechts';

		IF 	fb_trig_new_string.Q AND b_steuerung_ein THEN
			IF	s_tmp_string <> st_barcode_daten.s_band_anwahl AND
				s_tmp_string <> st_barcode_daten.s_band_ID_links AND
				b_bandende_rechts AND
				FIND(s_tmp_string,'-') <> 4 AND
				LEN(s_tmp_string) >8 AND
				(LEN(s_tmp_string) =10 OR gst_datensatz.st_md.i16_typ_zelle <> RASTERFOLIE) THEN
				st_barcode_daten.s_band_ID_rechts:=s_tmp_string;
				st_barcode_daten.b_band_ID_rechts_ok := TRUE;
				fb_tof_bm_neues_band_rechts.IN := TRUE;
				s_band_ID_rechtsHelp:=st_barcode_daten.s_band_ID_rechts;
			END_IF
			fb_state_entry.i16_next_step := BEREIT;
		END_IF

		(* Wartezeit abgelaufen => Wieder bereit *)
		IF 	fb_state_entry.fb_ton_Step.ET > t#5s THEN
 			fb_state_entry.s_debugtext:=CONCAT(fb_state_entry.s_debugtext,' => Wartezeit abgelaufen');
			fb_state_entry.i16_next_step := BEREIT;
		END_IF

(*=======================================================*)
	500:  fb_state_entry.s_debugtext:='Band 1720';

		IF 	fb_trig_new_string.Q THEN
			Anwahl();
			IF  	fb_state_entry.i16_next_step = 500  AND s_tmp_string = st_barcode_daten.s_band_anwahl AND b_bandende_1720 THEN
				st_barcode_daten.b_band_ok := TRUE;
				fb_tof_bm_neues_band_1720.IN := TRUE;
				fb_state_entry.i16_next_step := BEREIT;
			END_IF
		END_IF

		(* Wartezeit abgelaufen => Wieder bereit *)
		IF 	fb_state_entry.fb_ton_Step.ET > t#5s THEN
 			fb_state_entry.s_debugtext:=CONCAT(fb_state_entry.s_debugtext,' => Wartezeit abgelaufen');
			fb_state_entry.i16_next_step := BEREIT;
		END_IF

(*=======================================================*)
	STOP,FEHLER:

		IF	fb_state_entry.fb_ton_Step.ET > t#1s THEN
			fb_state_entry.i16_next_step := INIT;
		END_IF

END_CASE

fb_state_entry(i16_pos:= 2 );

(* Aufruf Baustein für serielle Kommunikation *)
fb_com_port_control(
	Mode:= SERIALLINEMODE_PC_COM_PORT,
	pComIn:= ADR(COM_in_data),			(* I/O data; see global variables *)
	pComOut:= ADR(COM_out_data),		(* I/O data; see global variables *)
	SizeComIn:= SIZEOF(COM_in_data),		(* I/O data; see global variables *)
	TxBuffer:= TxBuffer,					(* transmit buffer; see global variables *)
	RxBuffer:= RxBuffer,					(* receive buffer; see global variables *)
	Error=> com_port_control_error,
	ErrorID=> com_port_control_error_id);
(* =================================== *)

(* Routine für Strings empfangen *)
fb_receive(
	Timeout:= t#50ms,
	ReceivedString:= s_tmp_string,
	RXbuffer:= RxBuffer );

fb_trig_new_string(CLK:= fb_receive.StringReceived, Q=> );

(* Meldungs TOFs *)
fb_tof_bm_neues_band_links(IN:= , PT:= t#30s, Q=> , ET=> );
fb_tof_bm_neues_band_rechts(IN:= , PT:= t#30s, Q=> , ET=> );
fb_tof_bm_neues_band_1720(IN:= , PT:= t#30s, Q=> , ET=> );
fb_tof_bm_neues_wkz(IN:= , PT:= t#30s, Q=> , ET=> );

IF st_config.b_config_fertig THEN
	(* Fehlermeldungen ab dem Startindex in das globale Störmeldungsarray schreiben *)
	garr_stoermeldungen[st_config.i16_meld_startindex + 0] := sm_fehler_seriel;
	garr_stoermeldungen[st_config.i16_meld_startindex + 1] := FALSE;
	garr_stoermeldungen[st_config.i16_meld_startindex + 2] := FALSE;
	garr_stoermeldungen[st_config.i16_meld_startindex + 3] := FALSE;
	garr_stoermeldungen[st_config.i16_meld_startindex + 4] := FALSE;
	garr_stoermeldungen[st_config.i16_meld_startindex + 5] := FALSE;
	garr_stoermeldungen[st_config.i16_meld_startindex + 6] := FALSE;
	garr_stoermeldungen[st_config.i16_meld_startindex + 7] := FALSE;
	garr_stoermeldungen[st_config.i16_meld_startindex + 8] := FALSE;
	garr_stoermeldungen[st_config.i16_meld_startindex + 9] := FALSE;
	garr_stoermeldungen[st_config.i16_meld_startindex + 10] := FALSE;
	garr_stoermeldungen[st_config.i16_meld_startindex + 11] := FALSE;
	garr_stoermeldungen[st_config.i16_meld_startindex + 12] := FALSE;
	garr_stoermeldungen[st_config.i16_meld_startindex + 13] := FALSE;
	garr_stoermeldungen[st_config.i16_meld_startindex + 14] := FALSE;
	garr_stoermeldungen[st_config.i16_meld_startindex + 15] := FALSE;
	garr_stoermeldungen[st_config.i16_meld_startindex + 16] := FALSE;
	garr_stoermeldungen[st_config.i16_meld_startindex + 17] := FALSE;
	garr_stoermeldungen[st_config.i16_meld_startindex + 18] := FALSE;
	garr_stoermeldungen[st_config.i16_meld_startindex + 19] := FALSE;
	
	garr_betriebsmeldungen[st_config.i16_meld_startindex + 0] := fb_tof_bm_neues_band_links.Q;
	garr_betriebsmeldungen[st_config.i16_meld_startindex + 1] := fb_tof_bm_neues_band_rechts.Q;
	garr_betriebsmeldungen[st_config.i16_meld_startindex + 2] := fb_tof_bm_neues_band_1720.Q;
	garr_betriebsmeldungen[st_config.i16_meld_startindex + 3] := fb_tof_bm_neues_wkz.Q;
	garr_betriebsmeldungen[st_config.i16_meld_startindex + 4] := bm_band_nicht_gescannt_links;
	garr_betriebsmeldungen[st_config.i16_meld_startindex + 5] := bm_band_nicht_gescannt_rechts;
	garr_betriebsmeldungen[st_config.i16_meld_startindex + 6] := FALSE;
	garr_betriebsmeldungen[st_config.i16_meld_startindex + 7] := FALSE;
	garr_betriebsmeldungen[st_config.i16_meld_startindex + 8] := FALSE;
	garr_betriebsmeldungen[st_config.i16_meld_startindex + 9] := FALSE;
	garr_betriebsmeldungen[st_config.i16_meld_startindex + 10] := FALSE;
	garr_betriebsmeldungen[st_config.i16_meld_startindex + 11] := FALSE;
	garr_betriebsmeldungen[st_config.i16_meld_startindex + 12] := FALSE;
	garr_betriebsmeldungen[st_config.i16_meld_startindex + 13] := FALSE;
	garr_betriebsmeldungen[st_config.i16_meld_startindex + 14] := FALSE;
	garr_betriebsmeldungen[st_config.i16_meld_startindex + 15] := FALSE;
	garr_betriebsmeldungen[st_config.i16_meld_startindex + 16] := FALSE;
	garr_betriebsmeldungen[st_config.i16_meld_startindex + 17] := FALSE;
	garr_betriebsmeldungen[st_config.i16_meld_startindex + 18] := FALSE;
	garr_betriebsmeldungen[st_config.i16_meld_startindex + 19] := FALSE;
END_IF
END_FUNCTION_BLOCK
ACTION Anwahl:
(* Prüfe auf Start Werkzeug, Band Links, Band Rechts, Band *)
IF 	s_tmp_string = s_start_wkz THEN
	fb_state_entry.i16_next_step := 200;
ELSIF
	s_tmp_string = s_start_band_links THEN
	IF	NOT st_barcode_daten.b_band_links_ok THEN
		fb_state_entry.i16_next_step := 300;
	ELSIF NOT st_barcode_daten.b_band_ID_links_ok THEN
		fb_state_entry.i16_next_step := 350;
	END_IF
ELSIF
	s_tmp_string = s_start_band_rechts THEN
	IF	NOT st_barcode_daten.b_band_rechts_ok THEN
		fb_state_entry.i16_next_step := 400;
	ELSIF NOT st_barcode_daten.b_band_ID_rechts_ok THEN
		fb_state_entry.i16_next_step := 450;
	END_IF
ELSIF
	s_tmp_string = s_start_band THEN
	fb_state_entry.i16_next_step := 500;
END_IF
END_ACTION
ACTION ChargeToLTS:
(*	UML Nummer und VPE ermitteln,
	 diese werden mit einer Nummer auf die Pille geschrieben um Zeit zu sparen*)

(*gst_tag_data.UmlNo_VPE = erste Zahl immer 1 + UMl-Nummer max 99   danach max 6 Stellen für VPE => z.B.    1 78 100123 *)
st_LTS_xml.UmlNo:= STRING_TO_DINT(LEFT(DINT_TO_STRING(gst_tag_data.UmlNo_VPE),3))  - 100;		(*Uml Nummer => immer die ersten 3 Stellen -100 *)

i_actuellVPE:=	STRING_TO_DINT(		RIGHT(	DINT_TO_STRING(gst_tag_data.UmlNo_VPE), LEN(	DINT_TO_STRING(gst_tag_data.UmlNo_VPE)	)-3   ) 	);	(*VPE => die ersten 3 Stellen entfernen *)

(* ==================================Schrittkette============================================================================================ *)
fb_state_entry2(i16_pos:= 1);

CASE fb_state_entry2.i16_step OF
(*=======================================================*)
INIT_OBJ:

	IF	ST_BBGen.b_lesen_komplett THEN
		fb_state_entry2.i16_next_step := BEREIT;
	END_IF

(*=======================================================*)
BEREIT:  fb_state_entry2.s_debugtext:='Warte Ereigniss';

	IF	gst_PersDaten.st_LTS.i_tmpVPE <> i_actuellVPE AND
		i_actuellVPE <> 0 AND
		st_LTS_xml.UmlNo <> 0 AND   					  					(*beim Rüsten kann UML Nr. 0 auf die Pille geschrieben werden, dann wird nichts gebucht*)
		gst_datensatz.st_md.b_wt_transport_aktiv AND							(*damit beim Rüsten nicht gebucht wird*)
		gi16_maschinenstatusinfo = STATUS_MASCHINE_ARBEITET AND
		gst_datensatz.st_bestueckprogramm.i32_anzahl>0 AND
		(ST_Virtuelle_Masterachse.fb_state_entry.i16_step > BEREIT OR		(*Es darf nur gebucht werden, wenn auch tatsächlich bestückt wird*)
		ST_Rasterfolienmontage.fb_state_entry.i16_step > BEREIT ) THEN

		CASE gst_datensatz.st_md.i16_typ_zelle OF
		BESTUECKZELLE_1700:

			(*Bei 1700 wird die ID nur auf der linken Seite beschrieben da nur ein Band benutzt wird*)
			st_LTS_xml.newbatch[1]:='';							(*wird nur bei 1720 benutzt*)
			gst_PersDaten.st_LTS.s_tmpNewbatch[1]:='';			(*wird nur bei 1720 benutzt*)

			IF 	st_barcode_daten.b_band_ID_links_ok AND
				zyl_bandeinzuege_verschieben.st_ctrl.out.b_ausgefahren THEN
				st_LTS_xml.newbatch[0]:=st_barcode_daten.s_band_ID_links;
			ELSIF
				st_barcode_daten.b_band_ID_rechts_ok AND
				zyl_bandeinzuege_verschieben.st_ctrl.out.b_eingefahren THEN
				st_LTS_xml.newbatch[0]:=st_barcode_daten.s_band_ID_rechts;
			END_IF
			b_newbatchOk:=	st_LTS_xml.newbatch[0] <>'';								(*es muss ein Band eingescannt sein um eine Datei zu erstelle*)

		 RASTERFOLIE:

			(*Bei RASTERFOLIE wird die ID nur auf der linken Seite beschrieben da nur ein Band benutzt wird*)
			st_LTS_xml.newbatch[1]:='';							(*wird nur bei 1720 benutzt*)
			gst_PersDaten.st_LTS.s_tmpNewbatch[1]:='';			(*wird nur bei 1720 benutzt*)

			IF 	st_barcode_daten.b_band_ID_links_ok THEN
				st_LTS_xml.newbatch[0]:=st_barcode_daten.s_band_ID_links;
			END_IF
			b_newbatchOk:=	st_LTS_xml.newbatch[0] <>'';

		BESTUECKZELLE_1720:
			(*Bei 1720 wird die ID  auf beiden Seiten beschrieben da zwei Bänder gleichzeitig benutzt werden*)
			IF 	st_barcode_daten.b_band_ID_links_ok AND
			 	st_barcode_daten.b_band_ID_rechts_ok THEN
				st_LTS_xml.newbatch[0]:=st_barcode_daten.s_band_ID_links;
				st_LTS_xml.newbatch[1]:=st_barcode_daten.s_band_ID_rechts;
			END_IF
			b_newbatchOk:=st_LTS_xml.newbatch[0] <>'' AND st_LTS_xml.newbatch[1] <>'';		(*es müssen beide eingescannt sein um eine Datei zu erstelle*)

		END_CASE


		(*Trig startet das Erstellen der Xml und das Kopieren zum Server==========================================================*)
		IF 	b_newbatchOk THEN
			IF	(gst_PersDaten.st_LTS.i_tmpVPE > i_actuellVPE ) OR							(* bie einem neuen Auftrag*)
				((gst_PersDaten.st_LTS.s_tmpNewbatch[0] <> st_LTS_xml.newbatch[0]) 	AND st_LTS_xml.newbatch[0] <>'' ) OR	(* bei einer Äderung der Chargen ID*)
				((gst_PersDaten.st_LTS.s_tmpNewbatch[1] <> st_LTS_xml.newbatch[1])	AND st_LTS_xml.newbatch[1] <>'' ) THEN

				fb_state_entry2.i16_next_step := 110;
				gst_PersDaten.st_LTS.s_tmpNewbatch[0]:=st_LTS_xml.newbatch[0];
				gst_PersDaten.st_LTS.s_tmpNewbatch[1]:=st_LTS_xml.newbatch[1];
			END_IF
		END_IF

		gst_PersDaten.st_LTS.i_tmpVPE:=i_actuellVPE;

	END_IF

(*=======================================================*)
110:  fb_state_entry2.s_debugtext:='Dateinamen erstellen + VPE und Zeit in xml eintragen';

	IF	fb_state_entry2.E THEN

		st_LTS_xml.VPE:=i_actuellVPE;
		st_LTS_xml.timestamp:=gstr_system_time;

		s_FileName:='';
		s_FileName:=CONCAT(s_FileName, gst_datensatz.st_md.s_aktuelles_wkz);
		s_FileName:=CONCAT(s_FileName, '_');
		s_FileName:=CONCAT(s_FileName,WORD_TO_STR_LEN(gst_system_time.wDay,2));
		s_FileName:=CONCAT(s_FileName, '-');
		s_FileName:=CONCAT(s_FileName, WORD_TO_STR_LEN(gst_system_time.wMonth,2));
		s_FileName:=CONCAT(s_FileName, '-');
		s_FileName:=CONCAT(s_FileName, WORD_TO_STRING(gst_system_time.wYear));
		s_FileName:=CONCAT(s_FileName, '_');
		s_FileName:=CONCAT(s_FileName, WORD_TO_STR_LEN(gst_system_time.wHour,2));
		s_FileName:=CONCAT(s_FileName, '-');
		s_FileName:=CONCAT(s_FileName, WORD_TO_STR_LEN(gst_system_time.wMinute,2));
		s_FileName:=CONCAT(s_FileName, '-');
		s_FileName:=CONCAT(s_FileName, WORD_TO_STR_LEN(gst_system_time.wSecond,2));
		s_FileName:=CONCAT(s_FileName, '_');
		s_FileName:=CONCAT(s_FileName, st_LTS_xml.newbatch[0]);
		s_FileName:=CONCAT(s_FileName, '_');
		s_FileName:=CONCAT(s_FileName, DINT_TO_STRING(i_actuellVPE));
		s_FileName:=CONCAT(s_FileName, '.xml');
		fb_WriteXml.sFilePath :=CONCAT('D:\BBgen\LTS\',  s_FileName);
		fb_WriteXml.bExecute:=TRUE;

	END_IF

	IF	fb_WriteXml.bBusy THEN
		fb_state_entry2.i16_next_step := 120;
	ELSIF
		fb_WriteXml.bError THEN
		i_ErrId:= fb_WriteXml.nErrId;
		fb_state_entry2.i16_next_step := FEHLER;
	END_IF

	IF	fb_state_entry2.X THEN
		fb_WriteXml.bExecute:=FALSE;
	END_IF

(*=======================================================*)
120:  fb_state_entry2.s_debugtext:='warte auf fertig';

	IF	fb_state_entry2.fb_ton_Step.ET >t#500ms THEN
		IF	NOT fb_WriteXml.bBusy AND
			NOT fb_WriteXml.bError THEN
			fb_state_entry2.i16_next_step := 130;
		ELSIF
			fb_WriteXml.bError THEN
			i_ErrId:= fb_WriteXml.nErrId;
			fb_state_entry2.i16_next_step := FEHLER;
		END_IF
	END_IF

(*=======================================================*)
130:  fb_state_entry2.s_debugtext:='start vbs Skript => kopiert xml zum Server';

	IF	fb_state_entry2.E THEN
		NT_StartProcess.START:=TRUE;
	END_IF

	IF	NT_StartProcess.BUSY THEN
		fb_state_entry2.i16_next_step := 140;
	ELSIF
		NT_StartProcess.ERR THEN
		i_ErrId:= NT_StartProcess.ERRID;
		fb_state_entry2.i16_next_step := FEHLER;
	END_IF

	IF	fb_state_entry2.X THEN
		NT_StartProcess.START:=FALSE;
	END_IF

(*=======================================================*)
140:  fb_state_entry2.s_debugtext:='warte auf fertig';

	IF	NOT NT_StartProcess.BUSY AND
		NOT NT_StartProcess.ERR THEN
		fb_state_entry2.i16_next_step := BEREIT;
	ELSIF
		NT_StartProcess.ERR THEN
		i_ErrId:= NT_StartProcess.ERRID;
		fb_state_entry2.i16_next_step := FEHLER;
	END_IF

(*=======================================================*)
STOP,FEHLER:

	IF 	fb_state_entry2.E THEN
		IF	i_ErrId <> 0 THEN
		 	fb_state_entry2.s_debugtext:=CONCAT('nErrId = ', UDINT_TO_STRING(i_ErrId)	);
		END_IF
		i_ErrId:=0;
	END_IF

	(*-----------------------Weiterschaltbedingungen----------------------------*)
	IF	fb_state_entry2.fb_ton_Step.ET > t#1s THEN
		fb_state_entry2.i16_next_step := BEREIT;
	END_IF

END_CASE

fb_state_entry2(i16_pos:= 2 );


fb_WriteXml(
	ePath:= PATH_GENERIC ,
	nMode:= XMLSRV_ADDMISSING,
	sSymName:='.barcode.fb.st_LTS_xml',
	sXPath:=  '/data',
	tTimeout:= t#10s );


NT_StartProcess(
	PATHSTR:= 'C:\Windows\System32\wscript.exe',
	DIRNAME:=s_tools_path,
	COMNDLINE:=CONCAT(visu.s_akt_sprache,'_LTS_nach_server.vbs'),
	TMOUT:= DEFAULT_ADS_TIMEOUT);
END_ACTION
ACTION HandeingabeID:
fb_ton_band_ID(
	IN:= 	s_band_ID_linksHelp <> st_barcode_daten.s_band_ID_links OR
			s_band_ID_rechtsHelp <> st_barcode_daten.s_band_ID_rechts ,
	PT:=t#500ms , Q=>  , ET=> );


(*Handeingabe links=========================================*)
IF	st_barcode_daten.b_band_links_ok AND
	fb_ton_band_ID.Q THEN

		IF	LEN(st_barcode_daten.s_band_ID_links) < 8 THEN
			st_barcode_daten.s_band_ID_links:=s_band_ID_linksHelp;
		ELSE
			s_band_ID_linksHelp:=st_barcode_daten.s_band_ID_links;
			st_barcode_daten.b_band_ID_links_ok := TRUE;
		END_IF

END_IF



(*Handeingabe rechts=========================================*)
IF	st_barcode_daten.b_band_rechts_ok AND
	fb_ton_band_ID.Q THEN

		IF	LEN(st_barcode_daten.s_band_ID_rechts) < 8 THEN
			st_barcode_daten.s_band_ID_rechts:=s_band_ID_rechtsHelp;

		ELSE
			s_band_ID_rechtsHelp:=st_barcode_daten.s_band_ID_rechts;
			st_barcode_daten.b_band_ID_rechts_ok := TRUE;
		END_IF
END_IF
END_ACTION

(* POU Gemeinsamkeiten17xx/Haspel/Einfach/ST_Einfachhaspelkontroller, ST *)
FUNCTION_BLOCK ST_Einfachhaspelkontroller
VAR_INPUT
	t_wartezeit_bandende			: TIME;
	t_wartezeit_notabschaltung		: TIME;
	st_config						: struct_config;
	st_ctrl_in						: struct_ctrl_in;
	e_steuerung_ein				: BOOL;
END_VAR
VAR_IN_OUT
	st_visu						: struct_visu;
END_VAR
VAR_OUTPUT
	st_ctrl_out					: struct_ctrl_out;
END_VAR
VAR
	fb_ton_wz					: TON;
	fb_ton_uez					: TON;
	fb_ton_vz					: TON;
	fb_ton_vz_bandende			: TON;
	fb_ton_quitt					: TON;
	fb_state_entry					: ST_StateEntry;
	sm_haspel_nicht_bb			: BOOL := FALSE;
	sm_haspel_notaus 			: BOOL := FALSE;
	sm_haspel_notabschaltung		: BOOL := FALSE;
	bm_haspel_bandende			: BOOL := FALSE;
	e_haspelmotor_bb			AT %I* : BOOL;
	e_haspel_notaus				AT %I* : BOOL;
	e_haspel_bandende			AT %I* : BOOL;
	e_haspel_einschalten			AT %I* : BOOL;
	e_haspel_ausschalten			AT %I* : BOOL;
	a_motor						AT %Q* : BOOL;
END_VAR
(* Zeiten *)
fb_ton_wz(IN:= , PT:= , Q=>  , ET=> );
fb_ton_uez(IN:= , PT:= t_wartezeit_notabschaltung, Q=>  , ET=> );
fb_ton_vz(IN:= , PT:= t#5ms, Q=> , ET=> );
fb_ton_vz_bandende(IN:= e_haspel_bandende, PT:= t_wartezeit_bandende, Q=>  , ET=> );
fb_ton_quitt(IN:= , PT:= t#100ms, Q=> , ET=> );


(* Toplevel *)
IF fb_state_entry.i16_next_step > INIT AND fb_state_entry.i16_next_step < FEHLER THEN
	IF fb_state_entry.i16_next_step < STOP THEN
		IF st_ctrl_in.b_stop THEN
			fb_state_entry.i16_next_step := STOP;
		END_IF
	END_IF
	(* Allgemeine Fehler *)
	IF e_haspel_notaus THEN
		sm_haspel_notaus := TRUE;
		fb_state_entry.i16_next_step := FEHLER;
	ELSIF e_steuerung_ein AND NOT e_haspelmotor_bb THEN
		sm_haspel_nicht_bb := TRUE;
		fb_state_entry.i16_next_step := FEHLER;
	END_IF
	(* Bandende am Haspelbandeinzug *)
	IF fb_ton_vz_bandende.Q THEN
		bm_haspel_bandende := TRUE;
		st_ctrl_out.b_bandende := TRUE;
	ELSE
		IF e_haspel_ausschalten THEN
			bm_haspel_bandende := FALSE;
			st_ctrl_out.b_bandende := FALSE;
		END_IF
	END_IF
END_IF

(* ==================================Schrittkette================================ *)
fb_state_entry(
	i16_next_step:= ,
	i16_pos:= 1,
	s_debugtext:= ,
	E=> ,
	X=> , 
	i16_step=> ,
	i16_last_step=> );

CASE fb_state_entry.i16_step OF
(*=======================================================*)
	INIT_OBJ:
		IF st_config.b_config_fertig THEN
			fb_state_entry.i16_next_step := INIT;
		END_IF

(*=======================================================*)
	INIT:
		IF fb_state_entry.E THEN
			fb_ton_wz.IN := FALSE;
			fb_ton_uez.IN	:= FALSE;
			fb_ton_vz.IN := FALSE;
			fb_ton_quitt.IN := FALSE;
			sm_haspel_nicht_bb := FALSE;
			sm_haspel_notaus := FALSE;
			sm_haspel_notabschaltung := FALSE;
			bm_haspel_bandende	:= FALSE;
			st_ctrl_out.b_fehler := FALSE;
			st_ctrl_out.b_bereit := FALSE;
			st_ctrl_out.b_fertig := FALSE;
			st_ctrl_out.b_bandende := FALSE;
			a_motor := FALSE;
		END_IF

		(*-----------------------Weiterschaltbedingungen----------------------------*)
		IF st_ctrl_in.b_init THEN
			fb_state_entry.i16_next_step := BEREIT;
		END_IF

(*=======================================================*)
	BEREIT: (* Warte auf Sensor für Motor einschalten *)
		IF fb_state_entry.E THEN
			st_ctrl_out.b_bereit := TRUE;
			a_motor := FALSE;
		END_IF

		(*-----------------------Weiterschaltbedingungen----------------------------*)
		IF e_haspel_einschalten THEN
			fb_state_entry.i16_next_step := 110;
		END_IF

(*=======================================================*)
	110: (* Haspelmotor einschalten *)
		IF fb_state_entry.E THEN
			a_motor := TRUE;
			fb_ton_uez.IN := TRUE; (* Notabschaltung, weil etwas nicht stimmen kann *)
		END_IF

		(*-----------------------Weiterschaltbedingungen----------------------------*)
		IF e_haspel_ausschalten OR fb_ton_vz_bandende.Q THEN
			fb_ton_uez.IN := FALSE;
			fb_state_entry.i16_next_step := BEREIT;
		ELSIF fb_ton_uez.Q THEN
			fb_ton_uez.IN := FALSE;
			sm_haspel_notabschaltung := TRUE;
			fb_state_entry.i16_next_step := FEHLER;
		END_IF

(*=======================================================*)
	FEHLER:
		IF fb_state_entry.E THEN
			st_ctrl_out.b_fehler := TRUE;
			fb_ton_quitt.IN := FALSE;
			a_motor := FALSE;
		END_IF

		(*-----------------------Weiterschaltbedingungen----------------------------*)
		IF st_ctrl_in.b_quitt AND NOT fb_state_entry.E THEN
			st_ctrl_out.b_fehler := FALSE;
			fb_ton_quitt.IN := TRUE;
		END_IF

		IF fb_ton_quitt.Q THEN
			fb_ton_quitt.IN := FALSE;
			fb_state_entry.i16_next_step := INIT;
		END_IF

		(* Selbstquittierung, damit der Bediener das Band abspulen kann *)
		IF e_haspel_ausschalten THEN
			st_ctrl_out.b_fehler := FALSE;
			fb_ton_quitt.IN := FALSE;
			sm_haspel_nicht_bb := FALSE;
			sm_haspel_notaus := FALSE;
			sm_haspel_notabschaltung := FALSE;
			fb_state_entry.i16_next_step := 110;
		END_IF

(*=======================================================*)
	STOP:
		IF fb_state_entry.E THEN
			a_motor := FALSE;
			fb_ton_quitt.IN := FALSE;
		END_IF

		(*-----------------------Weiterschaltbedingungen----------------------------*)
		IF st_ctrl_in.b_quitt AND NOT fb_state_entry.E THEN
			fb_ton_quitt.IN := TRUE;
		END_IF

		IF fb_ton_quitt.Q THEN
			fb_ton_quitt.IN := FALSE;
			fb_state_entry.i16_next_step := INIT;
		END_IF
END_CASE

fb_state_entry(
	i16_next_step:= ,
	i16_pos:= 2,
	s_debugtext:= ,
	E=> , 
	X=> , 
	i16_step=> ,
	i16_last_step=> );

IF st_config.b_config_fertig THEN
	(* Fehlermeldungen und Betriebsmeldungen ab dem Startindex in die globalen Meldungsarrays schreiben *)
	garr_stoermeldungen[st_config.i16_meld_startindex + 0] := sm_haspel_notaus;
	garr_stoermeldungen[st_config.i16_meld_startindex + 1] := sm_haspel_nicht_bb;
	garr_stoermeldungen[st_config.i16_meld_startindex + 2] := sm_haspel_notabschaltung;
	garr_stoermeldungen[st_config.i16_meld_startindex + 3] := FALSE;
	garr_stoermeldungen[st_config.i16_meld_startindex + 4] := FALSE;
	garr_stoermeldungen[st_config.i16_meld_startindex + 5] := FALSE;
	garr_stoermeldungen[st_config.i16_meld_startindex + 6] := FALSE;
	garr_stoermeldungen[st_config.i16_meld_startindex + 7] := FALSE;
	garr_stoermeldungen[st_config.i16_meld_startindex + 8] := FALSE;
	garr_stoermeldungen[st_config.i16_meld_startindex + 9] := FALSE;
	garr_stoermeldungen[st_config.i16_meld_startindex + 10] := FALSE;
	garr_stoermeldungen[st_config.i16_meld_startindex + 11] := FALSE;
	garr_stoermeldungen[st_config.i16_meld_startindex + 12] := FALSE;
	garr_stoermeldungen[st_config.i16_meld_startindex + 13] := FALSE;
	garr_stoermeldungen[st_config.i16_meld_startindex + 14] := FALSE;
	garr_stoermeldungen[st_config.i16_meld_startindex + 15] := FALSE;
	garr_stoermeldungen[st_config.i16_meld_startindex + 16] := FALSE;
	garr_stoermeldungen[st_config.i16_meld_startindex + 17] := FALSE;
	garr_stoermeldungen[st_config.i16_meld_startindex + 18] := FALSE;
	garr_stoermeldungen[st_config.i16_meld_startindex + 19] := FALSE;
	
	garr_betriebsmeldungen[st_config.i16_meld_startindex + 0] := bm_haspel_bandende;
	garr_betriebsmeldungen[st_config.i16_meld_startindex + 1] := FALSE;
	garr_betriebsmeldungen[st_config.i16_meld_startindex + 2] := FALSE;
	garr_betriebsmeldungen[st_config.i16_meld_startindex + 3] := FALSE;
	garr_betriebsmeldungen[st_config.i16_meld_startindex + 4] := FALSE;
	garr_betriebsmeldungen[st_config.i16_meld_startindex + 5] := FALSE;
	garr_betriebsmeldungen[st_config.i16_meld_startindex + 6] := FALSE;
	garr_betriebsmeldungen[st_config.i16_meld_startindex + 7] := FALSE;
	garr_betriebsmeldungen[st_config.i16_meld_startindex + 8] := FALSE;
	garr_betriebsmeldungen[st_config.i16_meld_startindex + 9] := FALSE;
	garr_betriebsmeldungen[st_config.i16_meld_startindex + 10] := FALSE;
	garr_betriebsmeldungen[st_config.i16_meld_startindex + 11] := FALSE;
	garr_betriebsmeldungen[st_config.i16_meld_startindex + 12] := FALSE;
	garr_betriebsmeldungen[st_config.i16_meld_startindex + 13] := FALSE;
	garr_betriebsmeldungen[st_config.i16_meld_startindex + 14] := FALSE;
	garr_betriebsmeldungen[st_config.i16_meld_startindex + 15] := FALSE;
	garr_betriebsmeldungen[st_config.i16_meld_startindex + 16] := FALSE;
	garr_betriebsmeldungen[st_config.i16_meld_startindex + 17] := FALSE;
	garr_betriebsmeldungen[st_config.i16_meld_startindex + 18] := FALSE;
	garr_betriebsmeldungen[st_config.i16_meld_startindex + 19] := FALSE;
END_IF
END_FUNCTION_BLOCK

(* POU Gemeinsamkeiten17xx/Haspel/Einfach/ST_Haspel_V2, ST *)
FUNCTION_BLOCK ST_Haspel_V2
VAR_INPUT
	t_wartezeit_bandende			: TIME;
	st_config						: struct_config;
	st_ctrl_in						: struct_ctrl_in;
	b_bandende_Bandeinzug		: BOOL;
	b_band_ok					: BOOL;
END_VAR
VAR_IN_OUT
	st_visu						: struct_visu;
	st_zyl_heben				: struct_st_zylinder;
	st_zyl_abspulen				: struct_st_zylinder;
	st_zyl_sperren				: struct_st_zylinder;
END_VAR
VAR_OUTPUT
	st_ctrl_out					: struct_ctrl_out;
END_VAR
VAR
	fb_ton_wz					: TON;
	fb_ton_wz_bremse				: TON;
	fb_ton_uez					: TON;
	fb_ton_vz_einschalten			: TON;
	fb_ton_vz_bandende			: TON;
	fb_ton_bandende_Bandeinzug	: TON;
	fb_ton_quitt					: TON;
	fb_state_entry					: ST_StateEntry;
	sm_haspel_notaus 			: BOOL := FALSE;
	sm_haspel_notabschaltung		: BOOL := FALSE;
	bm_haspel_bandende			: BOOL := FALSE;
	e_haspel_notaus				AT %I* : BOOL;
	e_haspel_bandende			AT %I* : BOOL;
	e_haspel_einschalten			AT %I* : BOOL;
	e_haspel_ausschalten			AT %I* : BOOL;
END_VAR
(* Zeiten *)
fb_ton_wz(IN:= , PT:= , Q=>  , ET=> );
fb_ton_wz_bremse(IN:= , PT:= t#30s, Q=>  , ET=> );
fb_ton_uez(IN:= , PT:= t#15s, Q=>  , ET=> );
fb_ton_vz_einschalten(IN:= e_haspel_einschalten, PT:= t#50ms, Q=> , ET=> );
fb_ton_vz_bandende(IN:= e_haspel_bandende, PT:= t#1000ms, Q=>  , ET=> );
fb_ton_bandende_Bandeinzug(IN:=NOT b_bandende_Bandeinzug, PT:= t#1000ms, Q=>  , ET=> );
fb_ton_quitt(IN:= , PT:= t#50ms, Q=> , ET=> );

(* Toplevel *)
IF fb_state_entry.i16_next_step > INIT AND fb_state_entry.i16_next_step < FEHLER THEN
	(* Allgemeine Fehler *)
	IF e_haspel_notaus AND st_ctrl_in.b_freigabe THEN
		st_zyl_abspulen.st_ctrl.in.b_ausfahren := TRUE;
		sm_haspel_notaus := TRUE;
		fb_state_entry.i16_next_step := FEHLER;
	ELSIF 	st_zyl_heben.st_ctrl.out.b_fehler OR
			st_zyl_abspulen.st_ctrl.out.b_fehler OR
			st_zyl_sperren.st_ctrl.out.b_fehler
			THEN
				fb_state_entry.i16_next_step := FEHLER;
	ELSIF 	((st_visu.st_zyl.i16_nr_zyl_im_handbetrieb = st_zyl_heben.fb.st_config.i16_identnummer) OR
			(st_visu.st_zyl.i16_nr_zyl_im_handbetrieb = st_zyl_abspulen.fb.st_config.i16_identnummer) OR
			(st_visu.st_zyl.i16_nr_zyl_im_handbetrieb = st_zyl_sperren.fb.st_config.i16_identnummer)) AND
			gi16_betriebsart = HAND
			THEN
				fb_state_entry.i16_next_step := FEHLER;
	ELSE
		IF fb_state_entry.i16_next_step < STOP THEN
			IF st_ctrl_in.b_stop THEN
				st_zyl_abspulen.st_ctrl.in.b_ausfahren := TRUE;
				fb_state_entry.i16_next_step := STOP;
			END_IF
		END_IF
	END_IF

	(* Bandende am Haspelbandeinzug *)
	IF	 (gst_datensatz.st_md.i16_typ_zelle=BESTUECKZELLE_1700 OR
		gst_datensatz.st_md.i16_typ_zelle=RASTERFOLIE OR
		gst_datensatz.st_md.i16_typ_zelle=BESTUECKZELLE_1720) AND
		fb_ton_vz_bandende.Q AND st_ctrl_in.b_freigabe THEN
		bm_haspel_bandende := TRUE;
		st_ctrl_out.b_bandende := TRUE;
	ELSE
		bm_haspel_bandende := FALSE;
		st_ctrl_out.b_bandende := FALSE;
	END_IF
END_IF

(* ==================================Schrittkette================================ *)
fb_state_entry(
	i16_next_step:= ,
	i16_pos:= 1,
	s_debugtext:= ,
	E=> ,
	X=> , 
	i16_step=> ,
	i16_last_step=> );

CASE fb_state_entry.i16_step OF
(*=======================================================*)
	INIT_OBJ:
		IF st_config.b_config_fertig THEN
			fb_state_entry.i16_next_step := INIT;
		END_IF

(*=======================================================*)
	INIT:
		IF fb_state_entry.E THEN
			fb_ton_wz.IN := FALSE;
			fb_ton_wz_bremse.IN := FALSE;
			fb_ton_uez.IN := FALSE;
			fb_ton_vz_einschalten.IN := FALSE;
			fb_ton_quitt.IN := FALSE;
			sm_haspel_notaus := FALSE;
			sm_haspel_notabschaltung := FALSE;
			bm_haspel_bandende := FALSE;
			st_ctrl_out.b_fehler := FALSE;
			st_ctrl_out.b_bereit := FALSE;
			st_ctrl_out.b_fertig := FALSE;
			st_ctrl_out.b_bandende := FALSE;
			st_zyl_heben.st_ctrl.in.b_ausfahren := FALSE;
			st_zyl_heben.st_ctrl.in.b_einfahren := FALSE;
			st_zyl_abspulen.st_ctrl.in.b_ausfahren := FALSE;
			st_zyl_abspulen.st_ctrl.in.b_einfahren := FALSE;
			st_zyl_sperren.st_ctrl.in.b_ausfahren := FALSE;
			st_zyl_sperren.st_ctrl.in.b_einfahren := FALSE;
		END_IF

		(*-----------------------Weiterschaltbedingungen----------------------------*)
		IF st_ctrl_in.b_init THEN
			st_zyl_heben.st_ctrl.in.b_quittieren := FALSE;
			st_zyl_abspulen.st_ctrl.in.b_quittieren := FALSE;
			st_zyl_sperren.st_ctrl.in.b_quittieren := FALSE;
			fb_state_entry.i16_next_step := 20;
		END_IF

(*=======================================================*)
	20: (* Sperrzylinder ausfahren *)
		IF fb_state_entry.E THEN
			st_zyl_sperren.st_ctrl.in.b_ausfahren := TRUE;
		END_IF

		(*-----------------------Weiterschaltbedingungen----------------------------*)
		IF st_zyl_sperren.st_ctrl.out.b_ausgefahren AND st_ctrl_in.b_freigabe THEN
			fb_state_entry.i16_next_step := 30;
		ELSE
			fb_state_entry.i16_next_step := 40;
		END_IF

		IF fb_state_entry.X THEN
			st_zyl_sperren.st_ctrl.in.b_ausfahren := FALSE;
		END_IF

(*=======================================================*)
	30: (* Abspulzylinder ausfahren *)
		IF fb_state_entry.E THEN
			st_zyl_abspulen.st_ctrl.in.b_ausfahren := TRUE;
		END_IF

		(*-----------------------Weiterschaltbedingungen----------------------------*)
		IF st_zyl_abspulen.st_ctrl.out.b_ausgefahren THEN
			st_zyl_abspulen.st_ctrl.in.b_ausfahren := FALSE;
			fb_state_entry.i16_next_step := 40;
		END_IF

(*=======================================================*)
	40: (* Hebezylinder ausfahren *)
		IF fb_state_entry.E THEN
			st_zyl_heben.st_ctrl.in.b_ausfahren := TRUE;
		END_IF

		(*-----------------------Weiterschaltbedingungen----------------------------*)
		IF st_zyl_heben.st_ctrl.out.b_ausgefahren THEN
			st_zyl_heben.st_ctrl.in.b_ausfahren := FALSE;
			fb_state_entry.i16_next_step := BEREIT;
		END_IF

(*=======================================================*)
	BEREIT: (* Spule ist komplett angehoben und gesperrt, warte auf Sensor für einschalten *)
		IF fb_state_entry.E THEN
			sm_haspel_notaus := FALSE;
			st_ctrl_out.b_bereit := TRUE;
		END_IF

		CASE gst_datensatz.st_md.i16_typ_zelle OF

			KEINE_ZELLE:
				;

			BESTUECKZELLE_1700, RASTERFOLIE:
				(*-----------------------Weiterschaltbedingungen----------------------------*)
				IF st_ctrl_in.b_freigabe THEN(* Variable für aktive Seite, auf der abgespult wird *)
					(*bei Bandende die aktive Spule anheben*)
					IF e_haspel_einschalten THEN
						st_ctrl_out.b_kontroller_start := TRUE;
						fb_state_entry.i16_next_step := 110;
					ELSIF	(fb_ton_vz_bandende.Q OR fb_ton_bandende_Bandeinzug.Q) AND
					NOT st_zyl_abspulen.st_ctrl.out.b_ausgefahren THEN
						fb_state_entry.i16_next_step := 130;
					END_IF
				ELSE
					IF ST_Bandwechsel_Kontroller.b_spulenwechsel THEN
						IF NOT st_zyl_abspulen.st_ctrl.out.b_ausgefahren OR
						     fb_ton_bandende_Bandeinzug.Q THEN
							fb_state_entry.i16_next_step := 130;
						END_IF
					ELSE
						(* die nicht aktive Spule auf Bremse legen, wenn diese gesperrt wurde*)
						IF st_zyl_sperren.fb.e_sensor1_ausgefahren AND
						     NOT st_zyl_abspulen.st_ctrl.out.b_eingefahren THEN
							fb_state_entry.i16_next_step := 400;
						(* die nicht aktive Spule von Bremse heben, wenn diese freigegeben wurde*)
						ELSIF st_zyl_sperren.fb.e_sensor1_eingefahren AND
						     NOT st_zyl_abspulen.st_ctrl.out.b_ausgefahren THEN
							fb_state_entry.i16_next_step := 500;
						END_IF
					END_IF
				END_IF

			BESTUECKZELLE_1720:
				(*-----------------------Weiterschaltbedingungen----------------------------*)
				IF e_haspel_einschalten THEN
					st_ctrl_out.b_kontroller_start := TRUE;
					fb_state_entry.i16_next_step := 110;
				END_IF

		END_CASE

(*=======================================================*)
	110: (* Spule absenken und einschalten *)
		IF fb_state_entry.E THEN
			st_ctrl_out.b_kontroller_start := FALSE;
			bm_haspel_bandende := FALSE;
			st_ctrl_out.b_bandende := FALSE;
			st_zyl_abspulen.st_ctrl.in.b_einfahren := TRUE;
		END_IF

		(*-----------------------Weiterschaltbedingungen----------------------------*)
		IF st_zyl_abspulen.st_ctrl.out.b_eingefahren THEN
			st_zyl_abspulen.st_ctrl.in.b_einfahren := FALSE;
			fb_state_entry.i16_next_step := 120;
		END_IF

(*=======================================================*)
	120: (* Spule ist abgesenkt, warte auf Sensor für ausschalten *)
		IF fb_state_entry.E THEN
			fb_ton_uez.IN := TRUE; (* Notabschaltung, weil etwas nicht stimmen kann *)
		END_IF

		(*-----------------------Weiterschaltbedingungen----------------------------*)
		IF e_haspel_ausschalten OR
			gi16_betriebsart = HAND THEN	(* Wunsch von D. Rustler 07.04.22 dass auch im Handbetrieb der Haspel aufhört abzuspulen *)
			fb_ton_uez.IN := FALSE;
			fb_state_entry.i16_next_step := 130;
		ELSIF fb_ton_uez.Q THEN
			fb_ton_uez.IN := FALSE;
			sm_haspel_notabschaltung := TRUE;
			fb_state_entry.i16_next_step := 150;(* Spule anheben und dann in Fehler gehen *)
		END_IF

(*=======================================================*)
	130: (* Spule anheben *)
		IF fb_state_entry.E THEN
			st_zyl_abspulen.st_ctrl.in.b_ausfahren := TRUE;
		END_IF

		(*-----------------------Weiterschaltbedingungen----------------------------*)
		IF st_zyl_abspulen.st_ctrl.out.b_ausgefahren THEN
			st_zyl_abspulen.st_ctrl.in.b_ausfahren := FALSE;
			fb_state_entry.i16_next_step := BEREIT;
		ELSIF e_haspel_einschalten THEN
			st_zyl_abspulen.st_ctrl.in.b_ausfahren := FALSE;
			st_ctrl_out.b_kontroller_start := TRUE;
			fb_state_entry.i16_next_step := 110;
		END_IF

(*=======================================================*)
	150: (* Spule anheben und gehe in Fehler *)
		IF fb_state_entry.E THEN
			st_zyl_abspulen.st_ctrl.in.b_ausfahren := TRUE;
			fb_ton_wz.IN := TRUE;
			fb_ton_wz.PT := T#500ms;
		END_IF

		(*-----------------------Weiterschaltbedingungen----------------------------*)
		IF st_zyl_abspulen.st_ctrl.out.b_ausgefahren OR fb_ton_wz.Q THEN
			st_zyl_abspulen.st_ctrl.in.b_ausfahren := FALSE;
			fb_ton_wz.IN := FALSE;
			fb_state_entry.i16_next_step := FEHLER;
		END_IF

(*=======================================================*)
	400: (* Haspelspule auf Bremse legen 30 sek Wartezeit *)
		IF fb_state_entry.E THEN
			fb_ton_wz_bremse.IN := TRUE;
		END_IF

		(*-----------------------Weiterschaltbedingungen----------------------------*)
		IF fb_ton_wz_bremse.Q THEN
			fb_state_entry.i16_next_step := 410;
		END_IF

		IF fb_state_entry.X THEN
			fb_ton_wz_bremse.IN := FALSE;
		END_IF

(*=======================================================*)
	410: (* Haspelspule auf Bremse legen *)
		IF fb_state_entry.E THEN
			st_zyl_abspulen.st_ctrl.in.b_einfahren:=TRUE;
		END_IF

		(*-----------------------Weiterschaltbedingungen----------------------------*)
		IF st_zyl_abspulen.st_ctrl.out.b_eingefahren THEN
			st_zyl_abspulen.st_ctrl.in.b_einfahren:=FALSE;
			fb_state_entry.i16_next_step := BEREIT;
		END_IF

(*=======================================================*)
	500: (* Haspelspule von Bremse heben *)
		IF fb_state_entry.E THEN
			st_zyl_abspulen.st_ctrl.in.b_ausfahren:=TRUE;
		END_IF

		(*-----------------------Weiterschaltbedingungen----------------------------*)
		IF st_zyl_abspulen.st_ctrl.out.b_ausgefahren THEN
			st_zyl_abspulen.st_ctrl.in.b_ausfahren:=FALSE;
			fb_state_entry.i16_next_step := BEREIT;
		END_IF

(*=======================================================*)
	FEHLER:
		IF fb_state_entry.E THEN
			st_ctrl_out.b_fehler := TRUE;
			fb_ton_quitt.IN := FALSE;
			st_zyl_heben.st_ctrl.in.b_ausfahren := FALSE;
			st_zyl_heben.st_ctrl.in.b_einfahren := FALSE;
			st_zyl_abspulen.st_ctrl.in.b_ausfahren := FALSE;
			st_zyl_abspulen.st_ctrl.in.b_einfahren := FALSE;
			st_zyl_sperren.st_ctrl.in.b_ausfahren := FALSE;
			st_zyl_sperren.st_ctrl.in.b_einfahren := FALSE;
		END_IF

		(*Der Fehler Haspel Notaus, darf nur quittiert werden, wenn das Band ausgefädelt wurde*)
		IF sm_haspel_notaus AND NOT b_bandende_Bandeinzug THEN
			(*-----------------------Weiterschaltbedingungen----------------------------*)
			IF st_ctrl_in.b_quitt AND NOT fb_state_entry.E THEN
				st_ctrl_out.b_fehler := FALSE;
				st_zyl_heben.st_ctrl.in.b_quittieren := TRUE;
				st_zyl_abspulen.st_ctrl.in.b_quittieren := TRUE;
				st_zyl_sperren.st_ctrl.in.b_quittieren := TRUE;
				fb_ton_quitt.IN := TRUE;
			END_IF
		ELSIF NOT sm_haspel_notaus THEN
			(*-----------------------Weiterschaltbedingungen----------------------------*)
			IF st_ctrl_in.b_quitt AND NOT fb_state_entry.E THEN
				st_ctrl_out.b_fehler := FALSE;
				st_zyl_heben.st_ctrl.in.b_quittieren := TRUE;
				st_zyl_abspulen.st_ctrl.in.b_quittieren := TRUE;
				st_zyl_sperren.st_ctrl.in.b_quittieren := TRUE;
				fb_ton_quitt.IN := TRUE;
			END_IF
		END_IF

		IF fb_ton_quitt.Q THEN
			fb_ton_quitt.IN := FALSE;
			fb_state_entry.i16_next_step := INIT;
		END_IF

(*=======================================================*)
	STOP:
		IF fb_state_entry.E THEN
			st_ctrl_out.b_bereit := FALSE;
			fb_ton_quitt.IN := FALSE;
			st_zyl_heben.st_ctrl.in.b_ausfahren := FALSE;
			st_zyl_heben.st_ctrl.in.b_einfahren := FALSE;
			st_zyl_abspulen.st_ctrl.in.b_ausfahren := FALSE;
			st_zyl_abspulen.st_ctrl.in.b_einfahren := FALSE;
			st_zyl_sperren.st_ctrl.in.b_ausfahren := FALSE;
			st_zyl_sperren.st_ctrl.in.b_einfahren := FALSE;
		END_IF

		(*-----------------------Weiterschaltbedingungen----------------------------*)
		IF st_ctrl_in.b_quitt AND NOT fb_state_entry.E THEN
			fb_ton_quitt.IN := TRUE;
		END_IF

		IF fb_ton_quitt.Q THEN
			fb_ton_quitt.IN := FALSE;
			fb_state_entry.i16_next_step := INIT;
		END_IF
END_CASE

fb_state_entry(
	i16_next_step:= ,
	i16_pos:= 2,
	s_debugtext:= ,
	E=> , 
	X=> ,
	i16_step=> ,
	i16_last_step=> );

IF st_config.b_config_fertig THEN
	(* Fehlermeldungen und Betriebsmeldungen ab dem Startindex in die globalen Meldungsarrays schreiben *)
	garr_stoermeldungen[st_config.i16_meld_startindex + 0] := sm_haspel_notaus;
	garr_stoermeldungen[st_config.i16_meld_startindex + 1] := sm_haspel_notabschaltung;
	garr_stoermeldungen[st_config.i16_meld_startindex + 2] := FALSE;
	garr_stoermeldungen[st_config.i16_meld_startindex + 3] := FALSE;
	garr_stoermeldungen[st_config.i16_meld_startindex + 4] := FALSE;
	garr_stoermeldungen[st_config.i16_meld_startindex + 5] := FALSE;
	garr_stoermeldungen[st_config.i16_meld_startindex + 6] := FALSE;
	garr_stoermeldungen[st_config.i16_meld_startindex + 7] := FALSE;
	garr_stoermeldungen[st_config.i16_meld_startindex + 8] := FALSE;
	garr_stoermeldungen[st_config.i16_meld_startindex + 9] := FALSE;
	garr_stoermeldungen[st_config.i16_meld_startindex + 10] := FALSE;
	garr_stoermeldungen[st_config.i16_meld_startindex + 11] := FALSE;
	garr_stoermeldungen[st_config.i16_meld_startindex + 12] := FALSE;
	garr_stoermeldungen[st_config.i16_meld_startindex + 13] := FALSE;
	garr_stoermeldungen[st_config.i16_meld_startindex + 14] := FALSE;
	garr_stoermeldungen[st_config.i16_meld_startindex + 15] := FALSE;
	garr_stoermeldungen[st_config.i16_meld_startindex + 16] := FALSE;
	garr_stoermeldungen[st_config.i16_meld_startindex + 17] := FALSE;
	garr_stoermeldungen[st_config.i16_meld_startindex + 18] := FALSE;
	garr_stoermeldungen[st_config.i16_meld_startindex + 19] := FALSE;
	
	garr_betriebsmeldungen[st_config.i16_meld_startindex + 0] := bm_haspel_bandende;
	garr_betriebsmeldungen[st_config.i16_meld_startindex + 1] := FALSE;
	garr_betriebsmeldungen[st_config.i16_meld_startindex + 2] := FALSE;
	garr_betriebsmeldungen[st_config.i16_meld_startindex + 3] := FALSE;
	garr_betriebsmeldungen[st_config.i16_meld_startindex + 4] := FALSE;
	garr_betriebsmeldungen[st_config.i16_meld_startindex + 5] := FALSE;
	garr_betriebsmeldungen[st_config.i16_meld_startindex + 6] := FALSE;
	garr_betriebsmeldungen[st_config.i16_meld_startindex + 7] := FALSE;
	garr_betriebsmeldungen[st_config.i16_meld_startindex + 8] := FALSE;
	garr_betriebsmeldungen[st_config.i16_meld_startindex + 9] := FALSE;
	garr_betriebsmeldungen[st_config.i16_meld_startindex + 10] := FALSE;
	garr_betriebsmeldungen[st_config.i16_meld_startindex + 11] := FALSE;
	garr_betriebsmeldungen[st_config.i16_meld_startindex + 12] := FALSE;
	garr_betriebsmeldungen[st_config.i16_meld_startindex + 13] := FALSE;
	garr_betriebsmeldungen[st_config.i16_meld_startindex + 14] := FALSE;
	garr_betriebsmeldungen[st_config.i16_meld_startindex + 15] := FALSE;
	garr_betriebsmeldungen[st_config.i16_meld_startindex + 16] := FALSE;
	garr_betriebsmeldungen[st_config.i16_meld_startindex + 17] := FALSE;
	garr_betriebsmeldungen[st_config.i16_meld_startindex + 18] := FALSE;
	garr_betriebsmeldungen[st_config.i16_meld_startindex + 19] := FALSE;
END_IF
END_FUNCTION_BLOCK

(* POU Gemeinsamkeiten17xx/Haspel/ST_Haspel_st_zylinder, ST *)
FUNCTION_BLOCK ST_Haspel_st_zylinder
VAR_INPUT
	t_wartezeit_bandende			: TIME;
	e_druckwaechter				: BOOL;
	st_config						: struct_config;
	st_ctrl_in						: struct_ctrl_in;
END_VAR
VAR_IN_OUT
	st_visu						: struct_visu;
	st_zyl_heben					: struct_st_zylinder;
	st_zyl_sperren				: struct_st_zylinder;
END_VAR
VAR_OUTPUT
	st_ctrl_out					: struct_ctrl_out;
END_VAR
VAR
	fb_ton_wz					: TON;
	fb_ton_uez					: TON;
	fb_ton_vz					: TON;
	fb_ton_vz_bandende			: TON;
	fb_ton_quitt					: TON;
	fb_state_entry					: ST_StateEntry;
	sm_haspel_notaus 			: BOOL := FALSE;
	sm_haspel_notabschaltung		: BOOL := FALSE;
	bm_haspel_bandende			: BOOL := FALSE;
	e_haspel_notaus				AT %I* : BOOL;
	e_haspel_bandende			AT %I* : BOOL;
	e_haspel_einschalten			AT %I* : BOOL;
	e_haspel_ausschalten			AT %I* : BOOL;
END_VAR
(* Zeiten *)
fb_ton_wz(IN:= , PT:= , Q=>  , ET=> );
fb_ton_uez(IN:= , PT:= t#60s, Q=>  , ET=> );
fb_ton_vz(IN:= , PT:= t#100ms, Q=> , ET=> );
fb_ton_vz_bandende(IN:= e_haspel_bandende, PT:= t_wartezeit_bandende, Q=>  , ET=> );
fb_ton_quitt(IN:= , PT:= t#50ms, Q=> , ET=> );

(* Toplevel *)
IF fb_state_entry.i16_next_step > INIT AND fb_state_entry.i16_next_step < FEHLER THEN
	IF fb_state_entry.i16_next_step < STOP THEN
		IF st_ctrl_in.b_stop THEN
			st_zyl_heben.st_ctrl.in.b_ausfahren := TRUE;
			fb_state_entry.i16_next_step := STOP;
		END_IF
	END_IF
	(* Allgemeine Fehler *)
	IF e_haspel_notaus THEN
		st_zyl_heben.st_ctrl.in.b_ausfahren := TRUE;
		sm_haspel_notaus := TRUE;
		fb_state_entry.i16_next_step := FEHLER;
	ELSIF st_zyl_heben.st_ctrl.out.b_fehler OR st_zyl_sperren.st_ctrl.out.b_fehler THEN
		fb_state_entry.i16_next_step := FEHLER;
	ELSIF 	((st_visu.st_zyl.i16_nr_zyl_im_handbetrieb = st_zyl_heben.fb.st_config.i16_identnummer) OR
			(st_visu.st_zyl.i16_nr_zyl_im_handbetrieb = st_zyl_sperren.fb.st_config.i16_identnummer)) AND
			gi16_betriebsart = HAND
			THEN
			fb_state_entry.i16_next_step := FEHLER;
	END_IF

	(* Bandende am Haspelbandeinzug *)
	IF fb_ton_vz_bandende.Q THEN
		bm_haspel_bandende := st_ctrl_out.b_bandende := TRUE;
	ELSE
		bm_haspel_bandende := st_ctrl_out.b_bandende := FALSE;
	END_IF
END_IF

(* ==================================Schrittkette================================ *)
fb_state_entry(
	i16_next_step:= ,
	i16_pos:= 1,
	s_debugtext:= ,
	E=> ,
	X=> , 
	i16_step=> ,
	i16_last_step=> );

CASE fb_state_entry.i16_step OF
(*=======================================================*)
	INIT_OBJ:
		IF st_config.b_config_fertig THEN
			fb_state_entry.i16_next_step := INIT;
		END_IF

(*=======================================================*)
	INIT:
		IF fb_state_entry.E THEN
			fb_ton_wz.IN := FALSE;
			fb_ton_uez.IN	:= FALSE;
			fb_ton_vz.IN := FALSE;
			fb_ton_quitt.IN := FALSE;
			sm_haspel_notaus := FALSE;
			sm_haspel_notabschaltung := FALSE;
			bm_haspel_bandende	:= FALSE;
			st_ctrl_out.b_fehler := FALSE;
			st_ctrl_out.b_bereit := FALSE;
			st_ctrl_out.b_fertig := FALSE;
			st_ctrl_out.b_bandende := FALSE;
			st_zyl_heben.st_ctrl.in.b_ausfahren := FALSE;
			st_zyl_heben.st_ctrl.in.b_einfahren := FALSE;
			st_zyl_sperren.st_ctrl.in.b_ausfahren := FALSE;
			st_zyl_sperren.st_ctrl.in.b_einfahren := FALSE;
		END_IF

		(*-----------------------Weiterschaltbedingungen----------------------------*)
		IF st_ctrl_in.b_init THEN
			st_zyl_heben.st_ctrl.in.b_quittieren := FALSE;
			st_zyl_sperren.st_ctrl.in.b_quittieren := FALSE;
			fb_state_entry.i16_next_step := 20;
		END_IF

(*=======================================================*)
	20: (* Hebezylinder ausfahren *)
		IF fb_state_entry.E THEN
			st_zyl_heben.st_ctrl.in.b_ausfahren := TRUE;
		END_IF

		(*-----------------------Weiterschaltbedingungen----------------------------*)
		IF st_zyl_heben.st_ctrl.out.b_ausgefahren THEN
			st_zyl_heben.st_ctrl.in.b_ausfahren := FALSE;
			fb_state_entry.i16_next_step := 30;
		END_IF

(*=======================================================*)
	30: (* Sperrzylinder ausfahren *)
		IF fb_state_entry.E THEN
			st_zyl_sperren.st_ctrl.in.b_ausfahren := TRUE;
		END_IF

		(*-----------------------Weiterschaltbedingungen----------------------------*)
		IF st_zyl_sperren.st_ctrl.out.b_ausgefahren THEN
			st_zyl_sperren.st_ctrl.in.b_ausfahren := FALSE;
			fb_state_entry.i16_next_step := BEREIT;
		END_IF

(*=======================================================*)
	BEREIT: (* Spule ist angehoben und gesperrt, warte auf Sensor für einschalten *)
		IF fb_state_entry.E THEN
			st_ctrl_out.b_bereit := TRUE;
			st_ctrl_out.b_kontroller_start := FALSE;
		END_IF

		(*-----------------------Weiterschaltbedingungen----------------------------*)
		IF e_haspel_einschalten THEN
			st_ctrl_out.b_kontroller_start := TRUE;
			fb_state_entry.i16_next_step := 110;
		END_IF

(*=======================================================*)
	110: (* Spule absenken und einschalten *)
		IF fb_state_entry.E THEN
			st_zyl_heben.st_ctrl.in.b_einfahren := TRUE;
		END_IF

		(*-----------------------Weiterschaltbedingungen----------------------------*)
		IF st_zyl_heben.st_ctrl.out.b_eingefahren THEN
			st_zyl_heben.st_ctrl.in.b_einfahren := FALSE;
			fb_state_entry.i16_next_step := 120;
		END_IF

(*=======================================================*)
	120: (* Spule ist abgesenkt, warte auf Sensor für ausschalten *)
		IF fb_state_entry.E THEN
			fb_ton_uez.IN := TRUE; (* Notabschaltung, weil etwas nicht stimmen kann *)
		END_IF

		(*-----------------------Weiterschaltbedingungen----------------------------*)
		IF e_haspel_ausschalten THEN
			fb_ton_uez.IN := FALSE;
			fb_state_entry.i16_next_step := 130;
		ELSIF fb_ton_uez.Q THEN
			fb_ton_uez.IN := FALSE;
			sm_haspel_notabschaltung := TRUE;
			fb_state_entry.i16_next_step := FEHLER;
		END_IF

(*=======================================================*)
	130: (* Spule anheben und ausschalten *)
		IF fb_state_entry.E THEN
			st_zyl_heben.st_ctrl.in.b_ausfahren := TRUE;
		END_IF

		(*-----------------------Weiterschaltbedingungen----------------------------*)
		IF st_zyl_heben.st_ctrl.out.b_ausgefahren THEN
			st_zyl_heben.st_ctrl.in.b_ausfahren := FALSE;
			fb_state_entry.i16_next_step := BEREIT;
		END_IF

(*=======================================================*)
	FEHLER:
		IF fb_state_entry.E THEN
			st_ctrl_out.b_fehler := TRUE;
			fb_ton_quitt.IN := FALSE;
			st_ctrl_out.b_kontroller_start := FALSE;
			st_zyl_heben.st_ctrl.in.b_ausfahren := FALSE;
			st_zyl_heben.st_ctrl.in.b_einfahren := FALSE;
			st_zyl_sperren.st_ctrl.in.b_ausfahren := FALSE;
			st_zyl_sperren.st_ctrl.in.b_einfahren := FALSE;
		END_IF

		(*-----------------------Weiterschaltbedingungen----------------------------*)
		IF st_ctrl_in.b_quitt AND NOT fb_state_entry.E THEN
			st_ctrl_out.b_fehler := FALSE;
			st_zyl_heben.st_ctrl.in.b_quittieren := TRUE;
			st_zyl_sperren.st_ctrl.in.b_quittieren := TRUE;
			fb_ton_quitt.IN := TRUE;
		END_IF

		IF fb_ton_quitt.Q THEN
			fb_ton_quitt.IN := FALSE;
			fb_state_entry.i16_next_step := INIT;
		END_IF

(*=======================================================*)
	STOP:
		IF fb_state_entry.E THEN
			fb_ton_quitt.IN := FALSE;
			st_zyl_heben.st_ctrl.in.b_ausfahren := FALSE;
			st_zyl_heben.st_ctrl.in.b_einfahren := FALSE;
			st_zyl_sperren.st_ctrl.in.b_ausfahren := FALSE;
			st_zyl_sperren.st_ctrl.in.b_einfahren := FALSE;
		END_IF

		(*-----------------------Weiterschaltbedingungen----------------------------*)
		IF st_ctrl_in.b_quitt AND NOT fb_state_entry.E THEN
			fb_ton_quitt.IN := TRUE;
		END_IF

		IF fb_ton_quitt.Q THEN
			fb_ton_quitt.IN := FALSE;
			fb_state_entry.i16_next_step := INIT;
		END_IF
END_CASE

fb_state_entry(
	i16_next_step:= ,
	i16_pos:= 2,
	s_debugtext:= ,
	E=> , 
	X=> , 
	i16_step=> ,
	i16_last_step=> );

